LIN {X 0,Y 374.038,Z 429.773,A -85,B 0,C 180,E1 -12878.338,E2 -12878.338} C_VEL
LIN {X 0,Y 374.558,Z 418.473,A -85,B 0,C 180,E1 -12878.666,E2 -12878.666} C_VEL
LIN {X 0,Y 375.248,Z 375.181,A -85,B 0,C 180,E1 -12879.496,E2 -12879.496} C_VEL
LIN {X 0,Y 374.687,Z 369.374,A -85,B 0,C 180,E1 -12879.636,E2 -12879.636} C_VEL
LIN {X 0,Y 369.567,Z 350.642,A -85,B 0,C 180,E1 -12880.251,E2 -12880.251} C_VEL
LIN {X 0,Y 368.943,Z 344.836,A -85,B 0,C 180,E1 -12880.398,E2 -12880.398} C_VEL
LIN {X 0,Y 368.816,Z 338.494,A -85,B 0,C 180,E1 -12880.532,E2 -12880.532} C_VEL
LIN {X 0,Y 365.256,Z 319.525,A -85,B 0,C 180,E1 -12881.096,E2 -12881.096} C_VEL
LIN {X 0,Y 363.7,Z 314.51,A -85,B 0,C 180,E1 -12881.284,E2 -12881.284} C_VEL
LIN {X 0,Y 361.999,Z 305.393,A -85,B 0,C 180,E1 -12883.707,E2 -12883.707} C_VEL
LIN {X 0,Y 361.926,Z 305.399,A -85,B 0,C 180,E1 -12886.933,E2 -12886.933} C_VEL
LIN {X 0,Y 361.885,Z 305.41,A -85,B 0,C 180,E1 -12890.46,E2 -12890.46} C_VEL
LIN {X 0,Y 361.875,Z 305.406,A -85,B 0,C 180,E1 -12894.106,E2 -12894.106} C_VEL
LIN {X 0,Y 361.832,Z 305.41,A -85,B 0,C 180,E1 -12897.784,E2 -12897.784} C_VEL
LIN {X 0,Y 361.843,Z 305.41,A -85,B 0,C 180,E1 -12901.284,E2 -12901.284} C_VEL
LIN {X 0,Y 361.85,Z 305.409,A -85,B 0,C 180,E1 -12904.28,E2 -12904.28} C_VEL
LIN {X 0,Y 361.856,Z 305.41,A -85,B 0,C 180,E1 -12907.221,E2 -12907.221} C_VEL
LIN {X 0,Y 361.807,Z 305.417,A -85,B 0,C 180,E1 -12910.75,E2 -12910.75} C_VEL
LIN {X 0,Y 361.81,Z 305.413,A -85,B 0,C 180,E1 -12914.368,E2 -12914.368} C_VEL
LIN {X 0,Y 361.829,Z 305.413,A -85,B 0,C 180,E1 -12917.568,E2 -12917.568} C_VEL
LIN {X 0,Y 361.826,Z 305.414,A -85,B 0,C 180,E1 -12920.98,E2 -12920.98} C_VEL
LIN {X 0,Y 361.867,Z 305.406,A -85,B 0,C 180,E1 -12924.655,E2 -12924.655} C_VEL
LIN {X 0,Y 361.83,Z 305.41,A -85,B 0,C 180,E1 -12928.37,E2 -12928.37} C_VEL
LIN {X 0,Y 361.893,Z 305.403,A -85,B 0,C 180,E1 -12930.955,E2 -12930.955} C_VEL
LIN {X 0,Y 361.947,Z 305.401,A -85,B 0,C 180,E1 -12933.475,E2 -12933.475} C_VEL
LIN {X 0,Y 361.871,Z 305.406,A -85,B 0,C 180,E1 -12937.144,E2 -12937.144} C_VEL
LIN {X 0,Y 361.913,Z 305.399,A -85,B 0,C 180,E1 -12940.724,E2 -12940.724} C_VEL
LIN {X 0,Y 361.94,Z 305.399,A -85,B 0,C 180,E1 -12944.226,E2 -12944.226} C_VEL
LIN {X 0,Y 361.991,Z 305.391,A -85,B 0,C 180,E1 -12946.528,E2 -12946.528} C_VEL
LIN {X 0,Y 362.023,Z 305.391,A -85,B 0,C 180,E1 -12949.938,E2 -12949.938} C_VEL
LIN {X 0,Y 362.131,Z 305.372,A -85,B 0,C 180,E1 -12953.313,E2 -12953.313} C_VEL
LIN {X 0,Y 362.273,Z 305.357,A -85,B 0,C 180,E1 -12957.777,E2 -12957.777} C_VEL
LIN {X 0,Y 362.417,Z 305.34,A -85,B 0,C 180,E1 -12960,E2 -12960} C_VEL
LIN {X 0,Y 362.272,Z 305.36,A -85,B 0,C 180,E1 -12962.224,E2 -12962.224} C_VEL
LIN {X 0,Y 362.155,Z 305.374,A -85,B 0,C 180,E1 -12966.687,E2 -12966.687} C_VEL
LIN {X 0,Y 362.024,Z 305.387,A -85,B 0,C 180,E1 -12970.062,E2 -12970.062} C_VEL
LIN {X 0,Y 361.99,Z 305.39,A -85,B 0,C 180,E1 -12973.899,E2 -12973.899} C_VEL
LIN {X 0,Y 361.96,Z 305.394,A -85,B 0,C 180,E1 -12977.939,E2 -12977.939} C_VEL
LIN {X 0,Y 361.885,Z 305.403,A -85,B 0,C 180,E1 -12981.654,E2 -12981.654} C_VEL
LIN {X 0,Y 361.922,Z 305.402,A -85,B 0,C 180,E1 -12985.291,E2 -12985.291} C_VEL
LIN {X 0,Y 361.916,Z 305.399,A -85,B 0,C 180,E1 -12987.779,E2 -12987.779} C_VEL
LIN {X 0,Y 361.854,Z 305.409,A -85,B 0,C 180,E1 -12991.628,E2 -12991.628} C_VEL
LIN {X 0,Y 361.869,Z 305.411,A -85,B 0,C 180,E1 -12995.346,E2 -12995.346} C_VEL
LIN {X 0,Y 361.866,Z 305.408,A -85,B 0,C 180,E1 -12999.028,E2 -12999.028} C_VEL
LIN {X 0,Y 361.833,Z 305.41,A -85,B 0,C 180,E1 -13002.83,E2 -13002.83} C_VEL
LIN {X 0,Y 361.815,Z 305.414,A -85,B 0,C 180,E1 -13005.947,E2 -13005.947} C_VEL
LIN {X 0,Y 361.832,Z 305.412,A -85,B 0,C 180,E1 -13009.246,E2 -13009.246} C_VEL
LIN {X 0,Y 361.86,Z 305.406,A -85,B 0,C 180,E1 -13012.778,E2 -13012.778} C_VEL
LIN {X 0,Y 361.852,Z 305.413,A -85,B 0,C 180,E1 -13015.721,E2 -13015.721} C_VEL
LIN {X 0,Y 361.879,Z 305.408,A -85,B 0,C 180,E1 -13019.674,E2 -13019.674} C_VEL
LIN {X 0,Y 361.958,Z 305.54,A -85,B 0,C 180,E1 -13020.857,E2 -13020.857} C_VEL
LIN {X 0,Y 364.226,Z 316.996,A -85,B 0,C 180,E1 -13023.654,E2 -13023.654} C_VEL
LIN {X 0,Y 365.221,Z 322.463,A -85,B 0,C 180,E1 -13024.955,E2 -13024.955} C_VEL
LIN {X 0,Y 363.924,Z 338.418,A -85,B 0,C 180,E1 -13028.475,E2 -13028.475} C_VEL
LIN {X 0,Y 363.833,Z 339.649,A -85,B 0,C 180,E1 -13028.745,E2 -13028.745} C_VEL
LIN {X 0,Y 368.566,Z 373.996,A -85,B 0,C 180,E1 -13029.672,E2 -13029.672} C_VEL
LIN {X 0,Y 367.471,Z 448.258,A -85,B 0,C 180,E1 -13031.136,E2 -13031.136} C_VEL
LIN {X 0,Y 366.835,Z 461.529,A -85,B 0,C 180,E1 -13031.609,E2 -13031.609} C_VEL
LIN {X 0,Y 366.107,Z 473.727,A -85,B 0,C 180,E1 -13032.258,E2 -13032.258} C_VEL
LIN {X 0,Y 365.225,Z 485.208,A -85,B 0,C 180,E1 -13033.08,E2 -13033.08} C_VEL
LIN {X 0,Y 364.253,Z 497.008,A -85,B 0,C 180,E1 -13034.186,E2 -13034.186} C_VEL
LIN {X 0,Y 363.386,Z 507.607,A -85,B 0,C 180,E1 -13035.439,E2 -13035.439} C_VEL
LIN {X 0,Y 362.499,Z 517.133,A -85,B 0,C 180,E1 -13036.833,E2 -13036.833} C_VEL
LIN {X 0,Y 361.639,Z 526.297,A -85,B 0,C 180,E1 -13038.511,E2 -13038.511} C_VEL
LIN {X 0,Y 361.057,Z 533.678,A -85,B 0,C 180,E1 -13040.194,E2 -13040.194} C_VEL
LIN {X 0,Y 360.74,Z 538.672,A -85,B 0,C 180,E1 -13041.599,E2 -13041.599} C_VEL
LIN {X 0,Y 360.485,Z 543.511,A -85,B 0,C 180,E1 -13043.283,E2 -13043.283} C_VEL
LIN {X 0,Y 360.372,Z 547.214,A -85,B 0,C 180,E1 -13044.966,E2 -13044.966} C_VEL
LIN {X 0,Y 360.321,Z 549.885,A -85,B 0,C 180,E1 -13046.646,E2 -13046.646} C_VEL
LIN {X 0,Y 360.326,Z 551.141,A -85,B 0,C 180,E1 -13047.765,E2 -13047.765} C_VEL
LIN {X 0,Y 360.389,Z 551.991,A -85,B 0,C 180,E1 -13048.883,E2 -13048.883} C_VEL
LIN {X 0,Y 360.423,Z 552.4,A -85,B 0,C 180,E1 -13050.001,E2 -13050.001} C_VEL
LIN {X 0,Y 360.358,Z 552.415,A -85,B 0,C 180,E1 -13051.118,E2 -13051.118} C_VEL
LIN {X 0,Y 360.301,Z 551.289,A -85,B 0,C 180,E1 -13053.355,E2 -13053.355} C_VEL
LIN {X 0,Y 360.366,Z 550.094,A -85,B 0,C 180,E1 -13054.475,E2 -13054.475} C_VEL
LIN {X 0,Y 360.499,Z 546.471,A -85,B 0,C 180,E1 -13056.718,E2 -13056.718} C_VEL
LIN {X 0,Y 360.801,Z 542.572,A -85,B 0,C 180,E1 -13058.401,E2 -13058.401} C_VEL
LIN {X 0,Y 361.287,Z 537.56,A -85,B 0,C 180,E1 -13060.083,E2 -13060.083} C_VEL
LIN {X 0,Y 362.03,Z 531.286,A -85,B 0,C 180,E1 -13061.762,E2 -13061.762} C_VEL
LIN {X 0,Y 363.145,Z 523.46,A -85,B 0,C 180,E1 -13063.429,E2 -13063.429} C_VEL
LIN {X 0,Y 364.147,Z 515.494,A -85,B 0,C 180,E1 -13064.818,E2 -13064.818} C_VEL
LIN {X 0,Y 365.252,Z 505.819,A -85,B 0,C 180,E1 -13066.201,E2 -13066.201} C_VEL
LIN {X 0,Y 366.595,Z 495.078,A -85,B 0,C 180,E1 -13067.431,E2 -13067.431} C_VEL
LIN {X 0,Y 367.81,Z 484.646,A -85,B 0,C 180,E1 -13068.378,E2 -13068.378} C_VEL
LIN {X 0,Y 368.987,Z 472.123,A -85,B 0,C 180,E1 -13069.254,E2 -13069.254} C_VEL
LIN {X 0,Y 369.998,Z 458.92,A -85,B 0,C 180,E1 -13069.921,E2 -13069.921} C_VEL
LIN {X 0,Y 370.628,Z 446.91,A -85,B 0,C 180,E1 -13070.319,E2 -13070.319} C_VEL
LIN {X 0,Y 372.066,Z 375.094,A -85,B 0,C 180,E1 -13071.737,E2 -13071.737} C_VEL
LIN {X 0,Y 368.383,Z 353.004,A -85,B 0,C 180,E1 -13072.469,E2 -13072.469} C_VEL
LIN {X 0,Y 365.523,Z 339.056,A -85,B 0,C 180,E1 -13073.001,E2 -13073.001} C_VEL
LIN {X 0,Y 366.663,Z 327.943,A -85,B 0,C 180,E1 -13075.517,E2 -13075.517} C_VEL
LIN {X 0,Y 365.153,Z 319.279,A -85,B 0,C 180,E1 -13077.705,E2 -13077.705} C_VEL
LIN {X 0,Y 362.633,Z 308.581,A -85,B 0,C 180,E1 -13080.562,E2 -13080.562} C_VEL
LIN {X 0,Y 361.855,Z 305.416,A -85,B 0,C 180,E1 -13081.462,E2 -13081.462} C_VEL
LIN {X 0,Y 361.856,Z 305.415,A -85,B 0,C 180,E1 -13084.28,E2 -13084.28} C_VEL
LIN {X 0,Y 361.865,Z 305.41,A -85,B 0,C 180,E1 -13087.223,E2 -13087.223} C_VEL
LIN {X 0,Y 361.837,Z 305.414,A -85,B 0,C 180,E1 -13090.755,E2 -13090.755} C_VEL
LIN {X 0,Y 361.818,Z 305.415,A -85,B 0,C 180,E1 -13094.368,E2 -13094.368} C_VEL
LIN {X 0,Y 361.837,Z 305.41,A -85,B 0,C 180,E1 -13097.568,E2 -13097.568} C_VEL
LIN {X 0,Y 361.87,Z 305.411,A -85,B 0,C 180,E1 -13100.973,E2 -13100.973} C_VEL
LIN {X 0,Y 361.875,Z 305.409,A -85,B 0,C 180,E1 -13104.655,E2 -13104.655} C_VEL
LIN {X 0,Y 361.838,Z 305.411,A -85,B 0,C 180,E1 -13108.37,E2 -13108.37} C_VEL
LIN {X 0,Y 361.901,Z 305.404,A -85,B 0,C 180,E1 -13110.955,E2 -13110.955} C_VEL
LIN {X 0,Y 361.954,Z 305.395,A -85,B 0,C 180,E1 -13113.475,E2 -13113.475} C_VEL
LIN {X 0,Y 361.89,Z 305.402,A -85,B 0,C 180,E1 -13117.144,E2 -13117.144} C_VEL
LIN {X 0,Y 361.92,Z 305.398,A -85,B 0,C 180,E1 -13120.724,E2 -13120.724} C_VEL
LIN {X 0,Y 361.946,Z 305.394,A -85,B 0,C 180,E1 -13124.226,E2 -13124.226} C_VEL
LIN {X 0,Y 361.998,Z 305.385,A -85,B 0,C 180,E1 -13126.528,E2 -13126.528} C_VEL
LIN {X 0,Y 362.03,Z 305.38,A -85,B 0,C 180,E1 -13129.938,E2 -13129.938} C_VEL
LIN {X 0,Y 362.162,Z 305.368,A -85,B 0,C 180,E1 -13133.313,E2 -13133.313} C_VEL
LIN {X 0,Y 362.28,Z 305.353,A -85,B 0,C 180,E1 -13137.776,E2 -13137.776} C_VEL
LIN {X 0,Y 362.425,Z 305.332,A -85,B 0,C 180,E1 -13140,E2 -13140} C_VEL
LIN {X 0,Y 362.279,Z 305.351,A -85,B 0,C 180,E1 -13142.223,E2 -13142.223} C_VEL
LIN {X 0,Y 362.169,Z 305.364,A -85,B 0,C 180,E1 -13146.686,E2 -13146.686} C_VEL
LIN {X 0,Y 362.073,Z 305.379,A -85,B 0,C 180,E1 -13148.933,E2 -13148.933} C_VEL
LIN {X 0,Y 361.959,Z 305.392,A -85,B 0,C 180,E1 -13152.332,E2 -13152.332} C_VEL
LIN {X 0,Y 361.961,Z 305.398,A -85,B 0,C 180,E1 -13154.62,E2 -13154.62} C_VEL
LIN {X 0,Y 361.959,Z 305.395,A -85,B 0,C 180,E1 -13158.099,E2 -13158.099} C_VEL
LIN {X 0,Y 361.861,Z 305.405,A -85,B 0,C 180,E1 -13161.655,E2 -13161.655} C_VEL
LIN {X 0,Y 361.926,Z 305.399,A -85,B 0,C 180,E1 -13165.29,E2 -13165.29} C_VEL
LIN {X 0,Y 361.907,Z 305.396,A -85,B 0,C 180,E1 -13167.779,E2 -13167.779} C_VEL
LIN {X 0,Y 361.837,Z 305.406,A -85,B 0,C 180,E1 -13171.629,E2 -13171.629} C_VEL
LIN {X 0,Y 361.874,Z 305.406,A -85,B 0,C 180,E1 -13175.345,E2 -13175.345} C_VEL
LIN {X 0,Y 361.869,Z 305.41,A -85,B 0,C 180,E1 -13179.026,E2 -13179.026} C_VEL
LIN {X 0,Y 361.836,Z 305.411,A -85,B 0,C 180,E1 -13182.829,E2 -13182.829} C_VEL
LIN {X 0,Y 361.818,Z 305.415,A -85,B 0,C 180,E1 -13185.947,E2 -13185.947} C_VEL
LIN {X 0,Y 361.835,Z 305.414,A -85,B 0,C 180,E1 -13189.245,E2 -13189.245} C_VEL
LIN {X 0,Y 361.863,Z 305.406,A -85,B 0,C 180,E1 -13192.777,E2 -13192.777} C_VEL
LIN {X 0,Y 361.901,Z 305.436,A -85,B 0,C 180,E1 -13194.281,E2 -13194.281} C_VEL
LIN {X 0,Y 364.025,Z 314.87,A -85,B 0,C 180,E1 -13196.936,E2 -13196.936} C_VEL
LIN {X 0,Y 370.044,Z 329.595,A -85,B 0,C 180,E1 -13197.715,E2 -13197.715} C_VEL
LIN {X 0,Y 372.631,Z 341.079,A -85,B 0,C 180,E1 -13198.148,E2 -13198.148} C_VEL
LIN {X 0,Y 370.875,Z 421.936,A -85,B 0,C 180,E1 -13199.738,E2 -13199.738} C_VEL
LIN {X 0,Y 370.259,Z 434.827,A -85,B 0,C 180,E1 -13200.193,E2 -13200.193} C_VEL
LIN {X 0,Y 369.6,Z 447.003,A -85,B 0,C 180,E1 -13200.844,E2 -13200.844} C_VEL
LIN {X 0,Y 368.665,Z 458.851,A -85,B 0,C 180,E1 -13201.692,E2 -13201.692} C_VEL
LIN {X 0,Y 367.424,Z 470.91,A -85,B 0,C 180,E1 -13202.827,E2 -13202.827} C_VEL
LIN {X 0,Y 366.259,Z 481.223,A -85,B 0,C 180,E1 -13204.056,E2 -13204.056} C_VEL
LIN {X 0,Y 364.956,Z 491.237,A -85,B 0,C 180,E1 -13205.542,E2 -13205.542} C_VEL
LIN {X 0,Y 363.653,Z 500.421,A -85,B 0,C 180,E1 -13207.261,E2 -13207.261} C_VEL
LIN {X 0,Y 362.695,Z 507.766,A -85,B 0,C 180,E1 -13208.993,E2 -13208.993} C_VEL
LIN {X 0,Y 361.869,Z 513.554,A -85,B 0,C 180,E1 -13210.721,E2 -13210.721} C_VEL
LIN {X 0,Y 361.311,Z 517.926,A -85,B 0,C 180,E1 -13212.386,E2 -13212.386} C_VEL
LIN {X 0,Y 360.829,Z 521.454,A -85,B 0,C 180,E1 -13214.176,E2 -13214.176} C_VEL
LIN {X 0,Y 360.606,Z 523.12,A -85,B 0,C 180,E1 -13215.323,E2 -13215.323} C_VEL
LIN {X 0,Y 360.45,Z 524.885,A -85,B 0,C 180,E1 -13217.133,E2 -13217.133} C_VEL
LIN {X 0,Y 360.317,Z 525.591,A -85,B 0,C 180,E1 -13218.752,E2 -13218.752} C_VEL
LIN {X 0,Y 360.256,Z 525.204,A -85,B 0,C 180,E1 -13221.021,E2 -13221.021} C_VEL
LIN {X 0,Y 360.357,Z 524.401,A -85,B 0,C 180,E1 -13222.153,E2 -13222.153} C_VEL
LIN {X 0,Y 360.524,Z 522.465,A -85,B 0,C 180,E1 -13223.818,E2 -13223.818} C_VEL
LIN {X 0,Y 360.615,Z 519.498,A -85,B 0,C 180,E1 -13225.528,E2 -13225.528} C_VEL
LIN {X 0,Y 360.906,Z 515.533,A -85,B 0,C 180,E1 -13227.209,E2 -13227.209} C_VEL
LIN {X 0,Y 361.298,Z 509.444,A -85,B 0,C 180,E1 -13229.163,E2 -13229.163} C_VEL
LIN {X 0,Y 361.993,Z 502.786,A -85,B 0,C 180,E1 -13230.834,E2 -13230.834} C_VEL
LIN {X 0,Y 362.741,Z 494.551,A -85,B 0,C 180,E1 -13232.498,E2 -13232.498} C_VEL
LIN {X 0,Y 363.466,Z 486.104,A -85,B 0,C 180,E1 -13233.88,E2 -13233.88} C_VEL
LIN {X 0,Y 364.378,Z 475.674,A -85,B 0,C 180,E1 -13235.256,E2 -13235.256} C_VEL
LIN {X 0,Y 365.275,Z 466.727,A -85,B 0,C 180,E1 -13236.212,E2 -13236.212} C_VEL
LIN {X 0,Y 366.158,Z 455.721,A -85,B 0,C 180,E1 -13237.166,E2 -13237.166} C_VEL
LIN {X 0,Y 366.796,Z 443.576,A -85,B 0,C 180,E1 -13237.984,E2 -13237.984} C_VEL
LIN {X 0,Y 367.157,Z 430.842,A -85,B 0,C 180,E1 -13238.6,E2 -13238.6} C_VEL
LIN {X 0,Y 367.748,Z 418.549,A -85,B 0,C 180,E1 -13238.967,E2 -13238.967} C_VEL
LIN {X 0,Y 368.943,Z 344.836,A -85,B 0,C 180,E1 -13240.398,E2 -13240.398} C_VEL
LIN {X 0,Y 368.515,Z 340.992,A -85,B 0,C 180,E1 -13240.497,E2 -13240.497} C_VEL
LIN {X 0,Y 366.731,Z 335.502,A -85,B 0,C 180,E1 -13240.697,E2 -13240.697} C_VEL
LIN {X 0,Y 358.451,Z 320.029,A -85,B 0,C 180,E1 -13241.442,E2 -13241.442} C_VEL
LIN {X 0,Y 357.016,Z 316.361,A -85,B 0,C 180,E1 -13241.596,E2 -13241.596} C_VEL
LIN {X 0,Y 356.552,Z 314.673,A -85,B 0,C 180,E1 -13241.684,E2 -13241.684} C_VEL
LIN {X 0,Y 354.937,Z 306.273,A -85,B 0,C 180,E1 -13243.949,E2 -13243.949} C_VEL
LIN {X 0,Y 354.878,Z 306.276,A -85,B 0,C 180,E1 -13247.28,E2 -13247.28} C_VEL
LIN {X 0,Y 354.825,Z 306.285,A -85,B 0,C 180,E1 -13250.886,E2 -13250.886} C_VEL
LIN {X 0,Y 354.838,Z 306.288,A -85,B 0,C 180,E1 -13254.577,E2 -13254.577} C_VEL
LIN {X 0,Y 354.793,Z 306.29,A -85,B 0,C 180,E1 -13258.385,E2 -13258.385} C_VEL
LIN {X 0,Y 354.783,Z 306.29,A -85,B 0,C 180,E1 -13262.333,E2 -13262.333} C_VEL
LIN {X 0,Y 354.818,Z 306.283,A -85,B 0,C 180,E1 -13265.698,E2 -13265.698} C_VEL
LIN {X 0,Y 354.763,Z 306.292,A -85,B 0,C 180,E1 -13269.412,E2 -13269.412} C_VEL
LIN {X 0,Y 354.78,Z 306.293,A -85,B 0,C 180,E1 -13272.866,E2 -13272.866} C_VEL
LIN {X 0,Y 354.76,Z 306.29,A -85,B 0,C 180,E1 -13276.103,E2 -13276.103} C_VEL
LIN {X 0,Y 354.78,Z 306.294,A -85,B 0,C 180,E1 -13279.178,E2 -13279.178} C_VEL
LIN {X 0,Y 354.795,Z 306.286,A -85,B 0,C 180,E1 -13282.403,E2 -13282.403} C_VEL
LIN {X 0,Y 354.805,Z 306.287,A -85,B 0,C 180,E1 -13284.94,E2 -13284.94} C_VEL
LIN {X 0,Y 354.786,Z 306.287,A -85,B 0,C 180,E1 -13288.405,E2 -13288.405} C_VEL
LIN {X 0,Y 354.844,Z 306.286,A -85,B 0,C 180,E1 -13291.619,E2 -13291.619} C_VEL
LIN {X 0,Y 354.89,Z 306.276,A -85,B 0,C 180,E1 -13294.172,E2 -13294.172} C_VEL
LIN {X 0,Y 354.808,Z 306.289,A -85,B 0,C 180,E1 -13297.892,E2 -13297.892} C_VEL
LIN {X 0,Y 354.915,Z 306.277,A -85,B 0,C 180,E1 -13301.891,E2 -13301.891} C_VEL
LIN {X 0,Y 354.935,Z 306.275,A -85,B 0,C 180,E1 -13305.981,E2 -13305.981} C_VEL
LIN {X 0,Y 354.969,Z 306.268,A -85,B 0,C 180,E1 -13309.736,E2 -13309.736} C_VEL
LIN {X 0,Y 355.094,Z 306.249,A -85,B 0,C 180,E1 -13313.18,E2 -13313.18} C_VEL
LIN {X 0,Y 355.236,Z 306.233,A -85,B 0,C 180,E1 -13317.732,E2 -13317.732} C_VEL
LIN {X 0,Y 355.366,Z 306.218,A -85,B 0,C 180,E1 -13320,E2 -13320} C_VEL
LIN {X 0,Y 355.235,Z 306.237,A -85,B 0,C 180,E1 -13322.268,E2 -13322.268} C_VEL
LIN {X 0,Y 355.119,Z 306.249,A -85,B 0,C 180,E1 -13326.82,E2 -13326.82} C_VEL
LIN {X 0,Y 354.97,Z 306.267,A -85,B 0,C 180,E1 -13330.264,E2 -13330.264} C_VEL
LIN {X 0,Y 354.935,Z 306.269,A -85,B 0,C 180,E1 -13334.019,E2 -13334.019} C_VEL
LIN {X 0,Y 354.915,Z 306.272,A -85,B 0,C 180,E1 -13338.109,E2 -13338.109} C_VEL
LIN {X 0,Y 354.828,Z 306.282,A -85,B 0,C 180,E1 -13342.107,E2 -13342.107} C_VEL
LIN {X 0,Y 354.893,Z 306.274,A -85,B 0,C 180,E1 -13345.828,E2 -13345.828} C_VEL
LIN {X 0,Y 354.849,Z 306.281,A -85,B 0,C 180,E1 -13349.679,E2 -13349.679} C_VEL
LIN {X 0,Y 354.825,Z 306.284,A -85,B 0,C 180,E1 -13353.683,E2 -13353.683} C_VEL
LIN {X 0,Y 354.796,Z 306.286,A -85,B 0,C 180,E1 -13356.46,E2 -13356.46} C_VEL
LIN {X 0,Y 354.819,Z 306.289,A -85,B 0,C 180,E1 -13359.425,E2 -13359.425} C_VEL
LIN {X 0,Y 354.785,Z 306.289,A -85,B 0,C 180,E1 -13362.868,E2 -13362.868} C_VEL
LIN {X 0,Y 354.764,Z 306.291,A -85,B 0,C 180,E1 -13366.105,E2 -13366.105} C_VEL
LIN {X 0,Y 354.784,Z 306.29,A -85,B 0,C 180,E1 -13369.18,E2 -13369.18} C_VEL
LIN {X 0,Y 354.804,Z 306.286,A -85,B 0,C 180,E1 -13372.404,E2 -13372.404} C_VEL
LIN {X 0,Y 354.809,Z 306.285,A -85,B 0,C 180,E1 -13374.942,E2 -13374.942} C_VEL
LIN {X 0,Y 354.792,Z 306.288,A -85,B 0,C 180,E1 -13378.406,E2 -13378.406} C_VEL
LIN {X 0,Y 354.867,Z 306.307,A -85,B 0,C 180,E1 -13380.554,E2 -13380.554} C_VEL
LIN {X 0,Y 357.173,Z 317.74,A -85,B 0,C 180,E1 -13383.408,E2 -13383.408} C_VEL
LIN {X 0,Y 358.182,Z 323.116,A -85,B 0,C 180,E1 -13384.717,E2 -13384.717} C_VEL
LIN {X 0,Y 357.511,Z 332.543,A -85,B 0,C 180,E1 -13386.85,E2 -13386.85} C_VEL
LIN {X 0,Y 356.906,Z 339.368,A -85,B 0,C 180,E1 -13388.378,E2 -13388.378} C_VEL
LIN {X 0,Y 361.785,Z 374.313,A -85,B 0,C 180,E1 -13389.351,E2 -13389.351} C_VEL
LIN {X 0,Y 360.643,Z 448.305,A -85,B 0,C 180,E1 -13390.839,E2 -13390.839} C_VEL
LIN {X 0,Y 359.949,Z 462.24,A -85,B 0,C 180,E1 -13391.355,E2 -13391.355} C_VEL
LIN {X 0,Y 359.169,Z 474.728,A -85,B 0,C 180,E1 -13392.051,E2 -13392.051} C_VEL
LIN {X 0,Y 358.14,Z 487.459,A -85,B 0,C 180,E1 -13393.029,E2 -13393.029} C_VEL
LIN {X 0,Y 357.162,Z 498.792,A -85,B 0,C 180,E1 -13394.157,E2 -13394.157} C_VEL
LIN {X 0,Y 356.282,Z 508.981,A -85,B 0,C 180,E1 -13395.434,E2 -13395.434} C_VEL
LIN {X 0,Y 355.399,Z 518.164,A -85,B 0,C 180,E1 -13396.856,E2 -13396.856} C_VEL
LIN {X 0,Y 354.499,Z 527.105,A -85,B 0,C 180,E1 -13398.566,E2 -13398.566} C_VEL
LIN {X 0,Y 353.948,Z 534.277,A -85,B 0,C 180,E1 -13400.284,E2 -13400.284} C_VEL
LIN {X 0,Y 353.55,Z 539.983,A -85,B 0,C 180,E1 -13402.002,E2 -13402.002} C_VEL
LIN {X 0,Y 353.322,Z 545.136,A -85,B 0,C 180,E1 -13404.024,E2 -13404.024} C_VEL
LIN {X 0,Y 353.29,Z 547.863,A -85,B 0,C 180,E1 -13405.437,E2 -13405.437} C_VEL
LIN {X 0,Y 353.241,Z 549.542,A -85,B 0,C 180,E1 -13406.579,E2 -13406.579} C_VEL
LIN {X 0,Y 353.291,Z 551.691,A -85,B 0,C 180,E1 -13408.861,E2 -13408.861} C_VEL
LIN {X 0,Y 353.328,Z 552.126,A -85,B 0,C 180,E1 -13410.001,E2 -13410.001} C_VEL
LIN {X 0,Y 353.26,Z 552.159,A -85,B 0,C 180,E1 -13411.141,E2 -13411.141} C_VEL
LIN {X 0,Y 353.223,Z 551.071,A -85,B 0,C 180,E1 -13413.423,E2 -13413.423} C_VEL
LIN {X 0,Y 353.279,Z 549.906,A -85,B 0,C 180,E1 -13414.565,E2 -13414.565} C_VEL
LIN {X 0,Y 353.317,Z 547.907,A -85,B 0,C 180,E1 -13415.968,E2 -13415.968} C_VEL
LIN {X 0,Y 353.617,Z 543.886,A -85,B 0,C 180,E1 -13417.998,E2 -13417.998} C_VEL
LIN {X 0,Y 354.062,Z 539.299,A -85,B 0,C 180,E1 -13419.714,E2 -13419.714} C_VEL
LIN {X 0,Y 354.908,Z 532.378,A -85,B 0,C 180,E1 -13421.711,E2 -13421.711} C_VEL
LIN {X 0,Y 356.015,Z 524.91,A -85,B 0,C 180,E1 -13423.413,E2 -13423.413} C_VEL
LIN {X 0,Y 357.226,Z 515.93,A -85,B 0,C 180,E1 -13425.06,E2 -13425.06} C_VEL
LIN {X 0,Y 358.43,Z 506.023,A -85,B 0,C 180,E1 -13426.518,E2 -13426.518} C_VEL
LIN {X 0,Y 359.856,Z 495.385,A -85,B 0,C 180,E1 -13427.768,E2 -13427.768} C_VEL
LIN {X 0,Y 361.101,Z 485.113,A -85,B 0,C 180,E1 -13428.732,E2 -13428.732} C_VEL
LIN {X 0,Y 362.326,Z 472.876,A -85,B 0,C 180,E1 -13429.622,E2 -13429.622} C_VEL
LIN {X 0,Y 363.391,Z 460.031,A -85,B 0,C 180,E1 -13430.299,E2 -13430.299} C_VEL
LIN {X 0,Y 364.071,Z 447.666,A -85,B 0,C 180,E1 -13430.739,E2 -13430.739} C_VEL
LIN {X 0,Y 365.542,Z 375.302,A -85,B 0,C 180,E1 -13432.204,E2 -13432.204} C_VEL
LIN {X 0,Y 362.003,Z 354.385,A -85,B 0,C 180,E1 -13432.921,E2 -13432.921} C_VEL
LIN {X 0,Y 358.781,Z 338.808,A -85,B 0,C 180,E1 -13433.526,E2 -13433.526} C_VEL
LIN {X 0,Y 359.806,Z 329.05,A -85,B 0,C 180,E1 -13435.781,E2 -13435.781} C_VEL
LIN {X 0,Y 357.826,Z 318.845,A -85,B 0,C 180,E1 -13438.444,E2 -13438.444} C_VEL
LIN {X 0,Y 355.205,Z 307.939,A -85,B 0,C 180,E1 -13441.456,E2 -13441.456} C_VEL
LIN {X 0,Y 354.783,Z 306.296,A -85,B 0,C 180,E1 -13441.967,E2 -13441.967} C_VEL
LIN {X 0,Y 354.814,Z 306.288,A -85,B 0,C 180,E1 -13445.059,E2 -13445.059} C_VEL
LIN {X 0,Y 354.807,Z 306.291,A -85,B 0,C 180,E1 -13447.883,E2 -13447.883} C_VEL
LIN {X 0,Y 354.789,Z 306.291,A -85,B 0,C 180,E1 -13451.171,E2 -13451.171} C_VEL
LIN {X 0,Y 354.764,Z 306.293,A -85,B 0,C 180,E1 -13454.506,E2 -13454.506} C_VEL
LIN {X 0,Y 354.795,Z 306.287,A -85,B 0,C 180,E1 -13457.662,E2 -13457.662} C_VEL
LIN {X 0,Y 354.816,Z 306.285,A -85,B 0,C 180,E1 -13460.666,E2 -13460.666} C_VEL
LIN {X 0,Y 354.822,Z 306.284,A -85,B 0,C 180,E1 -13464.301,E2 -13464.301} C_VEL
LIN {X 0,Y 354.787,Z 306.289,A -85,B 0,C 180,E1 -13467.666,E2 -13467.666} C_VEL
LIN {X 0,Y 354.869,Z 306.277,A -85,B 0,C 180,E1 -13470.621,E2 -13470.621} C_VEL
LIN {X 0,Y 354.899,Z 306.273,A -85,B 0,C 180,E1 -13474.172,E2 -13474.172} C_VEL
LIN {X 0,Y 354.835,Z 306.282,A -85,B 0,C 180,E1 -13477.894,E2 -13477.894} C_VEL
LIN {X 0,Y 354.923,Z 306.27,A -85,B 0,C 180,E1 -13481.891,E2 -13481.891} C_VEL
LIN {X 0,Y 354.942,Z 306.265,A -85,B 0,C 180,E1 -13485.981,E2 -13485.981} C_VEL
LIN {X 0,Y 354.977,Z 306.259,A -85,B 0,C 180,E1 -13489.736,E2 -13489.736} C_VEL
LIN {X 0,Y 355.125,Z 306.243,A -85,B 0,C 180,E1 -13493.18,E2 -13493.18} C_VEL
LIN {X 0,Y 355.243,Z 306.23,A -85,B 0,C 180,E1 -13497.732,E2 -13497.732} C_VEL
LIN {X 0,Y 355.374,Z 306.21,A -85,B 0,C 180,E1 -13500,E2 -13500} C_VEL
LIN {X 0,Y 355.242,Z 306.227,A -85,B 0,C 180,E1 -13502.267,E2 -13502.267} C_VEL
LIN {X 0,Y 355.136,Z 306.239,A -85,B 0,C 180,E1 -13506.819,E2 -13506.819} C_VEL
LIN {X 0,Y 355.014,Z 306.257,A -85,B 0,C 180,E1 -13509.112,E2 -13509.112} C_VEL
LIN {X 0,Y 354.92,Z 306.269,A -85,B 0,C 180,E1 -13512.581,E2 -13512.581} C_VEL
LIN {X 0,Y 354.889,Z 306.275,A -85,B 0,C 180,E1 -13516.096,E2 -13516.096} C_VEL
LIN {X 0,Y 354.906,Z 306.277,A -85,B 0,C 180,E1 -13518.472,E2 -13518.472} C_VEL
LIN {X 0,Y 354.816,Z 306.284,A -85,B 0,C 180,E1 -13522.107,E2 -13522.107} C_VEL
LIN {X 0,Y 354.898,Z 306.273,A -85,B 0,C 180,E1 -13525.827,E2 -13525.827} C_VEL
LIN {X 0,Y 354.817,Z 306.283,A -85,B 0,C 180,E1 -13529.682,E2 -13529.682} C_VEL
LIN {X 0,Y 354.806,Z 306.284,A -85,B 0,C 180,E1 -13533.702,E2 -13533.702} C_VEL
LIN {X 0,Y 354.797,Z 306.288,A -85,B 0,C 180,E1 -13536.459,E2 -13536.459} C_VEL
LIN {X 0,Y 354.824,Z 306.285,A -85,B 0,C 180,E1 -13539.424,E2 -13539.424} C_VEL
LIN {X 0,Y 354.788,Z 306.289,A -85,B 0,C 180,E1 -13542.867,E2 -13542.867} C_VEL
LIN {X 0,Y 354.767,Z 306.293,A -85,B 0,C 180,E1 -13546.104,E2 -13546.104} C_VEL
LIN {X 0,Y 354.788,Z 306.292,A -85,B 0,C 180,E1 -13549.179,E2 -13549.179} C_VEL
LIN {X 0,Y 354.807,Z 306.283,A -85,B 0,C 180,E1 -13552.403,E2 -13552.403} C_VEL
LIN {X 0,Y 354.852,Z 306.332,A -85,B 0,C 180,E1 -13553.81,E2 -13553.81} C_VEL
LIN {X 0,Y 356.907,Z 315.288,A -85,B 0,C 180,E1 -13556.369,E2 -13556.369} C_VEL
LIN {X 0,Y 363.679,Z 331.28,A -85,B 0,C 180,E1 -13557.265,E2 -13557.265} C_VEL
LIN {X 0,Y 366.185,Z 342.113,A -85,B 0,C 180,E1 -13557.69,E2 -13557.69} C_VEL
LIN {X 0,Y 364.392,Z 422.475,A -85,B 0,C 180,E1 -13559.303,E2 -13559.303} C_VEL
LIN {X 0,Y 363.679,Z 436.04,A -85,B 0,C 180,E1 -13559.798,E2 -13559.798} C_VEL
LIN {X 0,Y 362.969,Z 448.613,A -85,B 0,C 180,E1 -13560.501,E2 -13560.501} C_VEL
LIN {X 0,Y 361.896,Z 460.862,A -85,B 0,C 180,E1 -13561.431,E2 -13561.431} C_VEL
LIN {X 0,Y 360.638,Z 472.576,A -85,B 0,C 180,E1 -13562.587,E2 -13562.587} C_VEL
LIN {X 0,Y 359.373,Z 482.784,A -85,B 0,C 180,E1 -13563.856,E2 -13563.856} C_VEL
LIN {X 0,Y 358.043,Z 492.37,A -85,B 0,C 180,E1 -13565.347,E2 -13565.347} C_VEL
LIN {X 0,Y 356.698,Z 501.403,A -85,B 0,C 180,E1 -13567.099,E2 -13567.099} C_VEL
LIN {X 0,Y 355.697,Z 508.603,A -85,B 0,C 180,E1 -13568.873,E2 -13568.873} C_VEL
LIN {X 0,Y 354.718,Z 515.061,A -85,B 0,C 180,E1 -13570.918,E2 -13570.918} C_VEL
LIN {X 0,Y 354.136,Z 519.287,A -85,B 0,C 180,E1 -13572.681,E2 -13572.681} C_VEL
LIN {X 0,Y 353.834,Z 521.5,A -85,B 0,C 180,E1 -13573.854,E2 -13573.854} C_VEL
LIN {X 0,Y 353.564,Z 523.209,A -85,B 0,C 180,E1 -13575.024,E2 -13575.024} C_VEL
LIN {X 0,Y 353.389,Z 525.161,A -85,B 0,C 180,E1 -13577.029,E2 -13577.029} C_VEL
LIN {X 0,Y 353.232,Z 525.839,A -85,B 0,C 180,E1 -13578.523,E2 -13578.523} C_VEL
LIN {X 0,Y 353.153,Z 525.529,A -85,B 0,C 180,E1 -13580.839,E2 -13580.839} C_VEL
LIN {X 0,Y 353.257,Z 524.789,A -85,B 0,C 180,E1 -13581.994,E2 -13581.994} C_VEL
LIN {X 0,Y 353.43,Z 522.697,A -85,B 0,C 180,E1 -13583.856,E2 -13583.856} C_VEL
LIN {X 0,Y 353.553,Z 518.84,A -85,B 0,C 180,E1 -13586.01,E2 -13586.01} C_VEL
LIN {X 0,Y 353.925,Z 514.595,A -85,B 0,C 180,E1 -13587.723,E2 -13587.723} C_VEL
LIN {X 0,Y 354.45,Z 508.18,A -85,B 0,C 180,E1 -13589.715,E2 -13589.715} C_VEL
LIN {X 0,Y 355.153,Z 501.148,A -85,B 0,C 180,E1 -13591.417,E2 -13591.417} C_VEL
LIN {X 0,Y 355.979,Z 492.39,A -85,B 0,C 180,E1 -13593.112,E2 -13593.112} C_VEL
LIN {X 0,Y 356.854,Z 482.456,A -85,B 0,C 180,E1 -13594.659,E2 -13594.659} C_VEL
LIN {X 0,Y 357.79,Z 472.286,A -85,B 0,C 180,E1 -13595.918,E2 -13595.918} C_VEL
LIN {X 0,Y 358.854,Z 462.522,A -85,B 0,C 180,E1 -13596.889,E2 -13596.889} C_VEL
LIN {X 0,Y 359.604,Z 450.278,A -85,B 0,C 180,E1 -13597.862,E2 -13597.862} C_VEL
LIN {X 0,Y 360.161,Z 438.668,A -85,B 0,C 180,E1 -13598.556,E2 -13598.556} C_VEL
LIN {X 0,Y 360.551,Z 427.29,A -85,B 0,C 180,E1 -13599.041,E2 -13599.041} C_VEL
LIN {X 0,Y 361.044,Z 413.744,A -85,B 0,C 180,E1 -13599.382,E2 -13599.382} C_VEL
LIN {X 0,Y 362.171,Z 340.065,A -85,B 0,C 180,E1 -13600.834,E2 -13600.834} C_VEL
LIN {X 0,Y 358.638,Z 321.225,A -85,B 0,C 180,E1 -13601.407,E2 -13601.407} C_VEL
LIN {X 0,Y 357.016,Z 316.361,A -85,B 0,C 180,E1 -13601.596,E2 -13601.596} C_VEL
LIN {X 0,Y 355.965,Z 314.814,A -85,B 0,C 180,E1 -13601.754,E2 -13601.754} C_VEL
LIN {X 0,Y 350.904,Z 311.687,A -85,B 0,C 180,E1 -13602.814,E2 -13602.814} C_VEL
LIN {X 0,Y 349.011,Z 309.812,A -85,B 0,C 180,E1 -13603.422,E2 -13603.422} C_VEL
LIN {X 0,Y 347.909,Z 307.271,A -85,B 0,C 180,E1 -13604.212,E2 -13604.212} C_VEL
LIN {X 0,Y 347.882,Z 307.153,A -85,B 0,C 180,E1 -13604.342,E2 -13604.342} C_VEL
LIN {X 0,Y 347.827,Z 307.159,A -85,B 0,C 180,E1 -13608.258,E2 -13608.258} C_VEL
LIN {X 0,Y 347.765,Z 307.162,A -85,B 0,C 180,E1 -13611.625,E2 -13611.625} C_VEL
LIN {X 0,Y 347.757,Z 307.164,A -85,B 0,C 180,E1 -13615.112,E2 -13615.112} C_VEL
LIN {X 0,Y 347.741,Z 307.168,A -85,B 0,C 180,E1 -13619.015,E2 -13619.015} C_VEL
LIN {X 0,Y 347.735,Z 307.166,A -85,B 0,C 180,E1 -13621.913,E2 -13621.913} C_VEL
LIN {X 0,Y 347.784,Z 307.16,A -85,B 0,C 180,E1 -13625.874,E2 -13625.874} C_VEL
LIN {X 0,Y 347.726,Z 307.172,A -85,B 0,C 180,E1 -13628.795,E2 -13628.795} C_VEL
LIN {X 0,Y 347.738,Z 307.165,A -85,B 0,C 180,E1 -13631.831,E2 -13631.831} C_VEL
LIN {X 0,Y 347.699,Z 307.176,A -85,B 0,C 180,E1 -13635.026,E2 -13635.026} C_VEL
LIN {X 0,Y 347.743,Z 307.165,A -85,B 0,C 180,E1 -13638.397,E2 -13638.397} C_VEL
LIN {X 0,Y 347.758,Z 307.163,A -85,B 0,C 180,E1 -13642.013,E2 -13642.013} C_VEL
LIN {X 0,Y 347.738,Z 307.17,A -85,B 0,C 180,E1 -13645.535,E2 -13645.535} C_VEL
LIN {X 0,Y 347.757,Z 307.168,A -85,B 0,C 180,E1 -13649.653,E2 -13649.653} C_VEL
LIN {X 0,Y 347.844,Z 307.152,A -85,B 0,C 180,E1 -13652.744,E2 -13652.744} C_VEL
LIN {X 0,Y 347.777,Z 307.162,A -85,B 0,C 180,E1 -13656.161,E2 -13656.161} C_VEL
LIN {X 0,Y 347.804,Z 307.162,A -85,B 0,C 180,E1 -13659.909,E2 -13659.909} C_VEL
LIN {X 0,Y 347.859,Z 307.152,A -85,B 0,C 180,E1 -13662.359,E2 -13662.359} C_VEL
LIN {X 0,Y 347.89,Z 307.153,A -85,B 0,C 180,E1 -13665.971,E2 -13665.971} C_VEL
LIN {X 0,Y 347.92,Z 307.144,A -85,B 0,C 180,E1 -13669.525,E2 -13669.525} C_VEL
LIN {X 0,Y 348.062,Z 307.125,A -85,B 0,C 180,E1 -13673.042,E2 -13673.042} C_VEL
LIN {X 0,Y 348.198,Z 307.109,A -85,B 0,C 180,E1 -13677.687,E2 -13677.687} C_VEL
LIN {X 0,Y 348.316,Z 307.096,A -85,B 0,C 180,E1 -13680,E2 -13680} C_VEL
LIN {X 0,Y 348.198,Z 307.114,A -85,B 0,C 180,E1 -13682.314,E2 -13682.314} C_VEL
LIN {X 0,Y 348.085,Z 307.124,A -85,B 0,C 180,E1 -13686.958,E2 -13686.958} C_VEL
LIN {X 0,Y 347.921,Z 307.148,A -85,B 0,C 180,E1 -13690.475,E2 -13690.475} C_VEL
LIN {X 0,Y 347.891,Z 307.148,A -85,B 0,C 180,E1 -13694.15,E2 -13694.15} C_VEL
LIN {X 0,Y 347.883,Z 307.149,A -85,B 0,C 180,E1 -13698.291,E2 -13698.291} C_VEL
LIN {X 0,Y 347.782,Z 307.16,A -85,B 0,C 180,E1 -13701.636,E2 -13701.636} C_VEL
LIN {X 0,Y 347.806,Z 307.162,A -85,B 0,C 180,E1 -13705.109,E2 -13705.109} C_VEL
LIN {X 0,Y 347.806,Z 307.158,A -85,B 0,C 180,E1 -13707.694,E2 -13707.694} C_VEL
LIN {X 0,Y 347.765,Z 307.162,A -85,B 0,C 180,E1 -13710.347,E2 -13710.347} C_VEL
LIN {X 0,Y 347.743,Z 307.165,A -85,B 0,C 180,E1 -13714.045,E2 -13714.045} C_VEL
LIN {X 0,Y 347.761,Z 307.169,A -85,B 0,C 180,E1 -13717.321,E2 -13717.321} C_VEL
LIN {X 0,Y 347.728,Z 307.167,A -85,B 0,C 180,E1 -13720.298,E2 -13720.298} C_VEL
LIN {X 0,Y 347.719,Z 307.174,A -85,B 0,C 180,E1 -13723.409,E2 -13723.409} C_VEL
LIN {X 0,Y 347.722,Z 307.167,A -85,B 0,C 180,E1 -13726.687,E2 -13726.687} C_VEL
LIN {X 0,Y 347.744,Z 307.166,A -85,B 0,C 180,E1 -13730.174,E2 -13730.174} C_VEL
LIN {X 0,Y 347.758,Z 307.163,A -85,B 0,C 180,E1 -13732.68,E2 -13732.68} C_VEL
LIN {X 0,Y 347.746,Z 307.169,A -85,B 0,C 180,E1 -13735.957,E2 -13735.957} C_VEL
LIN {X 0,Y 347.821,Z 307.16,A -85,B 0,C 180,E1 -13740.239,E2 -13740.239} C_VEL
LIN {X 0,Y 350.135,Z 318.466,A -85,B 0,C 180,E1 -13743.153,E2 -13743.153} C_VEL
LIN {X 0,Y 351.244,Z 324.897,A -85,B 0,C 180,E1 -13744.744,E2 -13744.744} C_VEL
LIN {X 0,Y 350.028,Z 339.056,A -85,B 0,C 180,E1 -13747.993,E2 -13747.993} C_VEL
LIN {X 0,Y 355.038,Z 375.372,A -85,B 0,C 180,E1 -13749.036,E2 -13749.036} C_VEL
LIN {X 0,Y 353.832,Z 448.266,A -85,B 0,C 180,E1 -13750.531,E2 -13750.531} C_VEL
LIN {X 0,Y 353.104,Z 462.128,A -85,B 0,C 180,E1 -13751.055,E2 -13751.055} C_VEL
LIN {X 0,Y 352.305,Z 474.572,A -85,B 0,C 180,E1 -13751.764,E2 -13751.764} C_VEL
LIN {X 0,Y 351.278,Z 486.479,A -85,B 0,C 180,E1 -13752.687,E2 -13752.687} C_VEL
LIN {X 0,Y 350.254,Z 498.077,A -85,B 0,C 180,E1 -13753.851,E2 -13753.851} C_VEL
LIN {X 0,Y 349.382,Z 507.776,A -85,B 0,C 180,E1 -13755.068,E2 -13755.068} C_VEL
LIN {X 0,Y 348.401,Z 517.538,A -85,B 0,C 180,E1 -13756.587,E2 -13756.587} C_VEL
LIN {X 0,Y 347.665,Z 525.178,A -85,B 0,C 180,E1 -13758.042,E2 -13758.042} C_VEL
LIN {X 0,Y 346.988,Z 532.662,A -85,B 0,C 180,E1 -13759.793,E2 -13759.793} C_VEL
LIN {X 0,Y 346.502,Z 539.544,A -85,B 0,C 180,E1 -13761.838,E2 -13761.838} C_VEL
LIN {X 0,Y 346.271,Z 544.197,A -85,B 0,C 180,E1 -13763.65,E2 -13763.65} C_VEL
LIN {X 0,Y 346.205,Z 547.502,A -85,B 0,C 180,E1 -13765.343,E2 -13765.343} C_VEL
LIN {X 0,Y 346.164,Z 549.2,A -85,B 0,C 180,E1 -13766.509,E2 -13766.509} C_VEL
LIN {X 0,Y 346.193,Z 551.385,A -85,B 0,C 180,E1 -13768.837,E2 -13768.837} C_VEL
LIN {X 0,Y 346.233,Z 551.853,A -85,B 0,C 180,E1 -13770.001,E2 -13770.001} C_VEL
LIN {X 0,Y 346.161,Z 551.902,A -85,B 0,C 180,E1 -13771.164,E2 -13771.164} C_VEL
LIN {X 0,Y 346.147,Z 550.849,A -85,B 0,C 180,E1 -13773.493,E2 -13773.493} C_VEL
LIN {X 0,Y 346.177,Z 549.717,A -85,B 0,C 180,E1 -13774.659,E2 -13774.659} C_VEL
LIN {X 0,Y 346.243,Z 547.944,A -85,B 0,C 180,E1 -13775.957,E2 -13775.957} C_VEL
LIN {X 0,Y 346.557,Z 543.761,A -85,B 0,C 180,E1 -13778.162,E2 -13778.162} C_VEL
LIN {X 0,Y 347.043,Z 539.218,A -85,B 0,C 180,E1 -13779.912,E2 -13779.912} C_VEL
LIN {X 0,Y 347.946,Z 532.362,A -85,B 0,C 180,E1 -13781.949,E2 -13781.949} C_VEL
LIN {X 0,Y 349.103,Z 524.951,A -85,B 0,C 180,E1 -13783.683,E2 -13783.683} C_VEL
LIN {X 0,Y 350.309,Z 516.344,A -85,B 0,C 180,E1 -13785.315,E2 -13785.315} C_VEL
LIN {X 0,Y 351.632,Z 506.243,A -85,B 0,C 180,E1 -13786.847,E2 -13786.847} C_VEL
LIN {X 0,Y 353.127,Z 495.705,A -85,B 0,C 180,E1 -13788.118,E2 -13788.118} C_VEL
LIN {X 0,Y 354.575,Z 483.956,A -85,B 0,C 180,E1 -13789.24,E2 -13789.24} C_VEL
LIN {X 0,Y 355.912,Z 471.386,A -85,B 0,C 180,E1 -13790.141,E2 -13790.141} C_VEL
LIN {X 0,Y 356.955,Z 458.875,A -85,B 0,C 180,E1 -13790.795,E2 -13790.795} C_VEL
LIN {X 0,Y 357.693,Z 445.859,A -85,B 0,C 180,E1 -13791.24,E2 -13791.24} C_VEL
LIN {X 0,Y 359.094,Z 375.72,A -85,B 0,C 180,E1 -13792.68,E2 -13792.68} C_VEL
LIN {X 0,Y 355.567,Z 355.359,A -85,B 0,C 180,E1 -13793.405,E2 -13793.405} C_VEL
LIN {X 0,Y 352.094,Z 338.431,A -85,B 0,C 180,E1 -13794.101,E2 -13794.101} C_VEL
LIN {X 0,Y 352.904,Z 330.472,A -85,B 0,C 180,E1 -13795.985,E2 -13795.985} C_VEL
LIN {X 0,Y 350.911,Z 320.185,A -85,B 0,C 180,E1 -13798.729,E2 -13798.729} C_VEL
LIN {X 0,Y 348.094,Z 308.639,A -85,B 0,C 180,E1 -13802.007,E2 -13802.007} C_VEL
LIN {X 0,Y 347.756,Z 307.166,A -85,B 0,C 180,E1 -13802.44,E2 -13802.44} C_VEL
LIN {X 0,Y 347.772,Z 307.168,A -85,B 0,C 180,E1 -13806.065,E2 -13806.065} C_VEL
LIN {X 0,Y 347.754,Z 307.168,A -85,B 0,C 180,E1 -13808.793,E2 -13808.793} C_VEL
LIN {X 0,Y 347.752,Z 307.168,A -85,B 0,C 180,E1 -13811.83,E2 -13811.83} C_VEL
LIN {X 0,Y 347.707,Z 307.173,A -85,B 0,C 180,E1 -13815.027,E2 -13815.027} C_VEL
LIN {X 0,Y 347.751,Z 307.168,A -85,B 0,C 180,E1 -13818.397,E2 -13818.397} C_VEL
LIN {X 0,Y 347.774,Z 307.162,A -85,B 0,C 180,E1 -13822.011,E2 -13822.011} C_VEL
LIN {X 0,Y 347.745,Z 307.162,A -85,B 0,C 180,E1 -13825.536,E2 -13825.536} C_VEL
LIN {X 0,Y 347.764,Z 307.16,A -85,B 0,C 180,E1 -13829.653,E2 -13829.653} C_VEL
LIN {X 0,Y 347.851,Z 307.153,A -85,B 0,C 180,E1 -13832.745,E2 -13832.745} C_VEL
LIN {X 0,Y 347.789,Z 307.159,A -85,B 0,C 180,E1 -13836.162,E2 -13836.162} C_VEL
LIN {X 0,Y 347.817,Z 307.156,A -85,B 0,C 180,E1 -13839.909,E2 -13839.909} C_VEL
LIN {X 0,Y 347.866,Z 307.148,A -85,B 0,C 180,E1 -13842.359,E2 -13842.359} C_VEL
LIN {X 0,Y 347.897,Z 307.142,A -85,B 0,C 180,E1 -13845.971,E2 -13845.971} C_VEL
LIN {X 0,Y 347.928,Z 307.138,A -85,B 0,C 180,E1 -13849.525,E2 -13849.525} C_VEL
LIN {X 0,Y 348.091,Z 307.119,A -85,B 0,C 180,E1 -13853.042,E2 -13853.042} C_VEL
LIN {X 0,Y 348.205,Z 307.106,A -85,B 0,C 180,E1 -13857.686,E2 -13857.686} C_VEL
LIN {X 0,Y 348.324,Z 307.088,A -85,B 0,C 180,E1 -13860,E2 -13860} C_VEL
LIN {X 0,Y 348.205,Z 307.103,A -85,B 0,C 180,E1 -13862.313,E2 -13862.313} C_VEL
LIN {X 0,Y 348.104,Z 307.115,A -85,B 0,C 180,E1 -13866.958,E2 -13866.958} C_VEL
LIN {X 0,Y 347.927,Z 307.144,A -85,B 0,C 180,E1 -13870.474,E2 -13870.474} C_VEL
LIN {X 0,Y 347.898,Z 307.148,A -85,B 0,C 180,E1 -13874.15,E2 -13874.15} C_VEL
LIN {X 0,Y 347.891,Z 307.149,A -85,B 0,C 180,E1 -13878.29,E2 -13878.29} C_VEL
LIN {X 0,Y 347.767,Z 307.161,A -85,B 0,C 180,E1 -13881.626,E2 -13881.626} C_VEL
LIN {X 0,Y 347.811,Z 307.156,A -85,B 0,C 180,E1 -13885.108,E2 -13885.108} C_VEL
LIN {X 0,Y 347.808,Z 307.153,A -85,B 0,C 180,E1 -13887.694,E2 -13887.694} C_VEL
LIN {X 0,Y 347.749,Z 307.165,A -85,B 0,C 180,E1 -13890.348,E2 -13890.348} C_VEL
LIN {X 0,Y 347.748,Z 307.163,A -85,B 0,C 180,E1 -13894.044,E2 -13894.044} C_VEL
LIN {X 0,Y 347.761,Z 307.163,A -85,B 0,C 180,E1 -13897.321,E2 -13897.321} C_VEL
LIN {X 0,Y 347.732,Z 307.164,A -85,B 0,C 180,E1 -13900.297,E2 -13900.297} C_VEL
LIN {X 0,Y 347.723,Z 307.172,A -85,B 0,C 180,E1 -13903.408,E2 -13903.408} C_VEL
LIN {X 0,Y 347.725,Z 307.169,A -85,B 0,C 180,E1 -13906.686,E2 -13906.686} C_VEL
LIN {X 0,Y 347.747,Z 307.168,A -85,B 0,C 180,E1 -13910.173,E2 -13910.173} C_VEL
LIN {X 0,Y 347.79,Z 307.328,A -85,B 0,C 180,E1 -13913.344,E2 -13913.344} C_VEL
LIN {X 0,Y 349.727,Z 315.435,A -85,B 0,C 180,E1 -13915.759,E2 -13915.759} C_VEL
LIN {X 0,Y 357.421,Z 333.257,A -85,B 0,C 180,E1 -13916.81,E2 -13916.81} C_VEL
LIN {X 0,Y 359.889,Z 343.711,A -85,B 0,C 180,E1 -13917.239,E2 -13917.239} C_VEL
LIN {X 0,Y 357.917,Z 422.992,A -85,B 0,C 180,E1 -13918.85,E2 -13918.85} C_VEL
LIN {X 0,Y 357.173,Z 436.474,A -85,B 0,C 180,E1 -13919.353,E2 -13919.353} C_VEL
LIN {X 0,Y 356.415,Z 449.223,A -85,B 0,C 180,E1 -13920.082,E2 -13920.082} C_VEL
LIN {X 0,Y 355.305,Z 461.214,A -85,B 0,C 180,E1 -13921.013,E2 -13921.013} C_VEL
LIN {X 0,Y 353.995,Z 472.912,A -85,B 0,C 180,E1 -13922.189,E2 -13922.189} C_VEL
LIN {X 0,Y 352.716,Z 482.735,A -85,B 0,C 180,E1 -13923.428,E2 -13923.428} C_VEL
LIN {X 0,Y 351.412,Z 491.848,A -85,B 0,C 180,E1 -13924.85,E2 -13924.85} C_VEL
LIN {X 0,Y 349.962,Z 501.013,A -85,B 0,C 180,E1 -13926.632,E2 -13926.632} C_VEL
LIN {X 0,Y 349.002,Z 507.622,A -85,B 0,C 180,E1 -13928.239,E2 -13928.239} C_VEL
LIN {X 0,Y 348.082,Z 513.243,A -85,B 0,C 180,E1 -13929.925,E2 -13929.925} C_VEL
LIN {X 0,Y 347.28,Z 518.611,A -85,B 0,C 180,E1 -13932.018,E2 -13932.018} C_VEL
LIN {X 0,Y 346.855,Z 521.523,A -85,B 0,C 180,E1 -13933.52,E2 -13933.52} C_VEL
LIN {X 0,Y 346.555,Z 523.3,A -85,B 0,C 180,E1 -13934.714,E2 -13934.714} C_VEL
LIN {X 0,Y 346.307,Z 525.449,A -85,B 0,C 180,E1 -13936.936,E2 -13936.936} C_VEL
LIN {X 0,Y 346.153,Z 526.083,A -85,B 0,C 180,E1 -13938.285,E2 -13938.285} C_VEL
LIN {X 0,Y 346.067,Z 525.854,A -85,B 0,C 180,E1 -13940.649,E2 -13940.649} C_VEL
LIN {X 0,Y 346.15,Z 525.154,A -85,B 0,C 180,E1 -13941.829,E2 -13941.829} C_VEL
LIN {X 0,Y 346.358,Z 522.973,A -85,B 0,C 180,E1 -13943.862,E2 -13943.862} C_VEL
LIN {X 0,Y 346.468,Z 519.402,A -85,B 0,C 180,E1 -13945.928,E2 -13945.928} C_VEL
LIN {X 0,Y 346.838,Z 515.246,A -85,B 0,C 180,E1 -13947.677,E2 -13947.677} C_VEL
LIN {X 0,Y 347.329,Z 508.928,A -85,B 0,C 180,E1 -13949.71,E2 -13949.71} C_VEL
LIN {X 0,Y 348.072,Z 502.041,A -85,B 0,C 180,E1 -13951.446,E2 -13951.446} C_VEL
LIN {X 0,Y 348.91,Z 493.427,A -85,B 0,C 180,E1 -13953.175,E2 -13953.175} C_VEL
LIN {X 0,Y 349.735,Z 484.616,A -85,B 0,C 180,E1 -13954.61,E2 -13954.61} C_VEL
LIN {X 0,Y 350.684,Z 474.929,A -85,B 0,C 180,E1 -13955.894,E2 -13955.894} C_VEL
LIN {X 0,Y 351.743,Z 465.686,A -85,B 0,C 180,E1 -13956.885,E2 -13956.885} C_VEL
LIN {X 0,Y 352.553,Z 454.334,A -85,B 0,C 180,E1 -13957.876,E2 -13957.876} C_VEL
LIN {X 0,Y 353.237,Z 441.349,A -85,B 0,C 180,E1 -13958.725,E2 -13958.725} C_VEL
LIN {X 0,Y 353.641,Z 429.199,A -85,B 0,C 180,E1 -13959.292,E2 -13959.292} C_VEL
LIN {X 0,Y 354.194,Z 417.035,A -85,B 0,C 180,E1 -13959.637,E2 -13959.637} C_VEL
LIN {X 0,Y 355.383,Z 340.651,A -85,B 0,C 180,E1 -13961.175,E2 -13961.175} C_VEL
LIN {X 0,Y 352.053,Z 323.083,A -85,B 0,C 180,E1 -13961.724,E2 -13961.724} C_VEL
LIN {X 0,Y 349.441,Z 315.049,A -85,B 0,C 180,E1 -13962.042,E2 -13962.042} C_VEL
LIN {X 0,Y 347.886,Z 307.153,A -85,B 0,C 180,E1 -13964.232,E2 -13964.232} C_VEL
LIN {X 0,Y 347.882,Z 307.153,A -85,B 0,C 180,E1 -13964.342,E2 -13964.342} C_VEL
LIN {X 0,Y 347.192,Z 307.234,A -85,B 0,C 180,E1 -13965.308,E2 -13965.308} C_VEL
LIN {X 0,Y 344.334,Z 307.591,A -85,B 0,C 180,E1 -13966.878,E2 -13966.878} C_VEL
LIN {X 0,Y 341.908,Z 307.895,A -85,B 0,C 180,E1 -13968.149,E2 -13968.149} C_VEL
LIN {X 0,Y 340.842,Z 308.026,A -85,B 0,C 180,E1 -13969.132,E2 -13969.132} C_VEL
LIN {X 0,Y 340.741,Z 308.037,A -85,B 0,C 180,E1 -13969.466,E2 -13969.466} C_VEL
LIN {X 0,Y 340.706,Z 308.043,A -85,B 0,C 180,E1 -13973.073,E2 -13973.073} C_VEL
LIN {X 0,Y 340.709,Z 308.041,A -85,B 0,C 180,E1 -13975.668,E2 -13975.668} C_VEL
LIN {X 0,Y 340.702,Z 308.042,A -85,B 0,C 180,E1 -13979.673,E2 -13979.673} C_VEL
LIN {X 0,Y 340.682,Z 308.047,A -85,B 0,C 180,E1 -13982.435,E2 -13982.435} C_VEL
LIN {X 0,Y 340.714,Z 308.043,A -85,B 0,C 180,E1 -13985.278,E2 -13985.278} C_VEL
LIN {X 0,Y 340.689,Z 308.044,A -85,B 0,C 180,E1 -13988.382,E2 -13988.382} C_VEL
LIN {X 0,Y 340.688,Z 308.043,A -85,B 0,C 180,E1 -13992.043,E2 -13992.043} C_VEL
LIN {X 0,Y 340.646,Z 308.049,A -85,B 0,C 180,E1 -13996.226,E2 -13996.226} C_VEL
LIN {X 0,Y 340.67,Z 308.047,A -85,B 0,C 180,E1 -13999.755,E2 -13999.755} C_VEL
LIN {X 0,Y 340.697,Z 308.048,A -85,B 0,C 180,E1 -14003.257,E2 -14003.257} C_VEL
LIN {X 0,Y 340.686,Z 308.044,A -85,B 0,C 180,E1 -14006.153,E2 -14006.153} C_VEL
LIN {X 0,Y 340.768,Z 308.033,A -85,B 0,C 180,E1 -14010.332,E2 -14010.332} C_VEL
LIN {X 0,Y 340.797,Z 308.031,A -85,B 0,C 180,E1 -14013.019,E2 -14013.019} C_VEL
LIN {X 0,Y 340.747,Z 308.043,A -85,B 0,C 180,E1 -14015.638,E2 -14015.638} C_VEL
LIN {X 0,Y 340.73,Z 308.041,A -85,B 0,C 180,E1 -14019.473,E2 -14019.473} C_VEL
LIN {X 0,Y 340.851,Z 308.028,A -85,B 0,C 180,E1 -14021.984,E2 -14021.984} C_VEL
LIN {X 0,Y 340.862,Z 308.026,A -85,B 0,C 180,E1 -14025.705,E2 -14025.705} C_VEL
LIN {X 0,Y 340.863,Z 308.021,A -85,B 0,C 180,E1 -14029.306,E2 -14029.306} C_VEL
LIN {X 0,Y 341.01,Z 308.004,A -85,B 0,C 180,E1 -14032.897,E2 -14032.897} C_VEL
LIN {X 0,Y 341.16,Z 307.986,A -85,B 0,C 180,E1 -14037.639,E2 -14037.639} C_VEL
LIN {X 0,Y 341.267,Z 307.974,A -85,B 0,C 180,E1 -14040,E2 -14040} C_VEL
LIN {X 0,Y 341.16,Z 307.99,A -85,B 0,C 180,E1 -14042.361,E2 -14042.361} C_VEL
LIN {X 0,Y 341.053,Z 307.999,A -85,B 0,C 180,E1 -14047.102,E2 -14047.102} C_VEL
LIN {X 0,Y 340.864,Z 308.026,A -85,B 0,C 180,E1 -14050.694,E2 -14050.694} C_VEL
LIN {X 0,Y 340.856,Z 308.025,A -85,B 0,C 180,E1 -14054.325,E2 -14054.325} C_VEL
LIN {X 0,Y 340.83,Z 308.029,A -85,B 0,C 180,E1 -14058.467,E2 -14058.467} C_VEL
LIN {X 0,Y 340.747,Z 308.036,A -85,B 0,C 180,E1 -14061.858,E2 -14061.858} C_VEL
LIN {X 0,Y 340.767,Z 308.034,A -85,B 0,C 180,E1 -14065.665,E2 -14065.665} C_VEL
LIN {X 0,Y 340.737,Z 308.038,A -85,B 0,C 180,E1 -14068.32,E2 -14068.32} C_VEL
LIN {X 0,Y 340.711,Z 308.046,A -85,B 0,C 180,E1 -14071.044,E2 -14071.044} C_VEL
LIN {X 0,Y 340.713,Z 308.047,A -85,B 0,C 180,E1 -14075.28,E2 -14075.28} C_VEL
LIN {X 0,Y 340.707,Z 308.041,A -85,B 0,C 180,E1 -14078.387,E2 -14078.387} C_VEL
LIN {X 0,Y 340.695,Z 308.044,A -85,B 0,C 180,E1 -14082.047,E2 -14082.047} C_VEL
LIN {X 0,Y 340.648,Z 308.049,A -85,B 0,C 180,E1 -14086.228,E2 -14086.228} C_VEL
LIN {X 0,Y 340.685,Z 308.049,A -85,B 0,C 180,E1 -14089.754,E2 -14089.754} C_VEL
LIN {X 0,Y 340.702,Z 308.044,A -85,B 0,C 180,E1 -14093.259,E2 -14093.259} C_VEL
LIN {X 0,Y 340.69,Z 308.047,A -85,B 0,C 180,E1 -14096.154,E2 -14096.154} C_VEL
LIN {X 0,Y 340.772,Z 308.195,A -85,B 0,C 180,E1 -14100.003,E2 -14100.003} C_VEL
LIN {X 0,Y 343.076,Z 319.192,A -85,B 0,C 180,E1 -14102.885,E2 -14102.885} C_VEL
LIN {X 0,Y 344.268,Z 326.032,A -85,B 0,C 180,E1 -14104.616,E2 -14104.616} C_VEL
LIN {X 0,Y 343.131,Z 338.82,A -85,B 0,C 180,E1 -14107.61,E2 -14107.61} C_VEL
LIN {X 0,Y 348.276,Z 376.11,A -85,B 0,C 180,E1 -14108.702,E2 -14108.702} C_VEL
LIN {X 0,Y 347.025,Z 448.194,A -85,B 0,C 180,E1 -14110.21,E2 -14110.21} C_VEL
LIN {X 0,Y 346.272,Z 461.991,A -85,B 0,C 180,E1 -14110.744,E2 -14110.744} C_VEL
LIN {X 0,Y 345.447,Z 474.394,A -85,B 0,C 180,E1 -14111.466,E2 -14111.466} C_VEL
LIN {X 0,Y 344.311,Z 487.078,A -85,B 0,C 180,E1 -14112.479,E2 -14112.479} C_VEL
LIN {X 0,Y 343.271,Z 498.388,A -85,B 0,C 180,E1 -14113.65,E2 -14113.65} C_VEL
LIN {X 0,Y 342.276,Z 509.214,A -85,B 0,C 180,E1 -14115.078,E2 -14115.078} C_VEL
LIN {X 0,Y 341.305,Z 518.546,A -85,B 0,C 180,E1 -14116.606,E2 -14116.606} C_VEL
LIN {X 0,Y 340.367,Z 527.322,A -85,B 0,C 180,E1 -14118.387,E2 -14118.387} C_VEL
LIN {X 0,Y 339.791,Z 534.318,A -85,B 0,C 180,E1 -14120.176,E2 -14120.176} C_VEL
LIN {X 0,Y 339.335,Z 540.729,A -85,B 0,C 180,E1 -14122.264,E2 -14122.264} C_VEL
LIN {X 0,Y 339.14,Z 545.028,A -85,B 0,C 180,E1 -14124.104,E2 -14124.104} C_VEL
LIN {X 0,Y 339.105,Z 547.134,A -85,B 0,C 180,E1 -14125.245,E2 -14125.245} C_VEL
LIN {X 0,Y 339.088,Z 548.855,A -85,B 0,C 180,E1 -14126.436,E2 -14126.436} C_VEL
LIN {X 0,Y 339.096,Z 551.076,A -85,B 0,C 180,E1 -14128.813,E2 -14128.813} C_VEL
LIN {X 0,Y 339.137,Z 551.578,A -85,B 0,C 180,E1 -14130.001,E2 -14130.001} C_VEL
LIN {X 0,Y 339.063,Z 551.646,A -85,B 0,C 180,E1 -14131.188,E2 -14131.188} C_VEL
LIN {X 0,Y 339.072,Z 550.628,A -85,B 0,C 180,E1 -14133.566,E2 -14133.566} C_VEL
LIN {X 0,Y 339.08,Z 549.529,A -85,B 0,C 180,E1 -14134.756,E2 -14134.756} C_VEL
LIN {X 0,Y 339.142,Z 547.983,A -85,B 0,C 180,E1 -14135.948,E2 -14135.948} C_VEL
LIN {X 0,Y 339.397,Z 544.891,A -85,B 0,C 180,E1 -14137.736,E2 -14137.736} C_VEL
LIN {X 0,Y 339.826,Z 540.758,A -85,B 0,C 180,E1 -14139.524,E2 -14139.524} C_VEL
LIN {X 0,Y 340.638,Z 534.463,A -85,B 0,C 180,E1 -14141.605,E2 -14141.605} C_VEL
LIN {X 0,Y 341.769,Z 527.634,A -85,B 0,C 180,E1 -14143.376,E2 -14143.376} C_VEL
LIN {X 0,Y 343.052,Z 519.149,A -85,B 0,C 180,E1 -14145.142,E2 -14145.142} C_VEL
LIN {X 0,Y 344.303,Z 510.45,A -85,B 0,C 180,E1 -14146.605,E2 -14146.605} C_VEL
LIN {X 0,Y 345.902,Z 499.765,A -85,B 0,C 180,E1 -14148.05,E2 -14148.05} C_VEL
LIN {X 0,Y 347.348,Z 489.144,A -85,B 0,C 180,E1 -14149.196,E2 -14149.196} C_VEL
LIN {X 0,Y 348.794,Z 477.278,A -85,B 0,C 180,E1 -14150.186,E2 -14150.186} C_VEL
LIN {X 0,Y 349.924,Z 464.973,A -85,B 0,C 180,E1 -14150.963,E2 -14150.963} C_VEL
LIN {X 0,Y 350.926,Z 452.322,A -85,B 0,C 180,E1 -14151.515,E2 -14151.515} C_VEL
LIN {X 0,Y 351.43,Z 437.415,A -85,B 0,C 180,E1 -14151.907,E2 -14151.907} C_VEL
LIN {X 0,Y 352.72,Z 376.934,A -85,B 0,C 180,E1 -14153.154,E2 -14153.154} C_VEL
LIN {X 0,Y 349.425,Z 357.515,A -85,B 0,C 180,E1 -14153.861,E2 -14153.861} C_VEL
LIN {X 0,Y 345.429,Z 338.175,A -85,B 0,C 180,E1 -14154.671,E2 -14154.671} C_VEL
LIN {X 0,Y 346.04,Z 333.099,A -85,B 0,C 180,E1 -14155.891,E2 -14155.891} C_VEL
LIN {X 0,Y 345.079,Z 326.668,A -85,B 0,C 180,E1 -14157.602,E2 -14157.602} C_VEL
LIN {X 0,Y 342.737,Z 316.234,A -85,B 0,C 180,E1 -14160.544,E2 -14160.544} C_VEL
LIN {X 0,Y 340.7,Z 308.042,A -85,B 0,C 180,E1 -14163.005,E2 -14163.005} C_VEL
LIN {X 0,Y 340.706,Z 308.045,A -85,B 0,C 180,E1 -14166.742,E2 -14166.742} C_VEL
LIN {X 0,Y 340.689,Z 308.047,A -85,B 0,C 180,E1 -14170.247,E2 -14170.247} C_VEL
LIN {X 0,Y 340.653,Z 308.052,A -85,B 0,C 180,E1 -14173.773,E2 -14173.773} C_VEL
LIN {X 0,Y 340.7,Z 308.043,A -85,B 0,C 180,E1 -14177.954,E2 -14177.954} C_VEL
LIN {X 0,Y 340.733,Z 308.039,A -85,B 0,C 180,E1 -14181.772,E2 -14181.772} C_VEL
LIN {X 0,Y 340.723,Z 308.036,A -85,B 0,C 180,E1 -14185.595,E2 -14185.595} C_VEL
LIN {X 0,Y 340.704,Z 308.042,A -85,B 0,C 180,E1 -14188.956,E2 -14188.956} C_VEL
LIN {X 0,Y 340.778,Z 308.034,A -85,B 0,C 180,E1 -14192.474,E2 -14192.474} C_VEL
LIN {X 0,Y 340.756,Z 308.038,A -85,B 0,C 180,E1 -14195.638,E2 -14195.638} C_VEL
LIN {X 0,Y 340.749,Z 308.04,A -85,B 0,C 180,E1 -14199.474,E2 -14199.474} C_VEL
LIN {X 0,Y 340.858,Z 308.022,A -85,B 0,C 180,E1 -14201.984,E2 -14201.984} C_VEL
LIN {X 0,Y 340.869,Z 308.017,A -85,B 0,C 180,E1 -14205.705,E2 -14205.705} C_VEL
LIN {X 0,Y 340.87,Z 308.018,A -85,B 0,C 180,E1 -14209.306,E2 -14209.306} C_VEL
LIN {X 0,Y 341.059,Z 307.994,A -85,B 0,C 180,E1 -14212.898,E2 -14212.898} C_VEL
LIN {X 0,Y 341.167,Z 307.984,A -85,B 0,C 180,E1 -14217.639,E2 -14217.639} C_VEL
LIN {X 0,Y 341.275,Z 307.965,A -85,B 0,C 180,E1 -14220,E2 -14220} C_VEL
LIN {X 0,Y 341.167,Z 307.979,A -85,B 0,C 180,E1 -14222.361,E2 -14222.361} C_VEL
LIN {X 0,Y 341.074,Z 307.99,A -85,B 0,C 180,E1 -14227.102,E2 -14227.102} C_VEL
LIN {X 0,Y 340.87,Z 308.021,A -85,B 0,C 180,E1 -14230.694,E2 -14230.694} C_VEL
LIN {X 0,Y 340.863,Z 308.026,A -85,B 0,C 180,E1 -14234.325,E2 -14234.325} C_VEL
LIN {X 0,Y 340.837,Z 308.03,A -85,B 0,C 180,E1 -14238.467,E2 -14238.467} C_VEL
LIN {X 0,Y 340.717,Z 308.039,A -85,B 0,C 180,E1 -14241.842,E2 -14241.842} C_VEL
LIN {X 0,Y 340.771,Z 308.033,A -85,B 0,C 180,E1 -14245.664,E2 -14245.664} C_VEL
LIN {X 0,Y 340.728,Z 308.034,A -85,B 0,C 180,E1 -14248.321,E2 -14248.321} C_VEL
LIN {X 0,Y 340.697,Z 308.041,A -85,B 0,C 180,E1 -14251.045,E2 -14251.045} C_VEL
LIN {X 0,Y 340.717,Z 308.04,A -85,B 0,C 180,E1 -14255.279,E2 -14255.279} C_VEL
LIN {X 0,Y 340.709,Z 308.042,A -85,B 0,C 180,E1 -14258.386,E2 -14258.386} C_VEL
LIN {X 0,Y 340.699,Z 308.044,A -85,B 0,C 180,E1 -14262.045,E2 -14262.045} C_VEL
LIN {X 0,Y 340.652,Z 308.051,A -85,B 0,C 180,E1 -14266.227,E2 -14266.227} C_VEL
LIN {X 0,Y 340.688,Z 308.048,A -85,B 0,C 180,E1 -14269.753,E2 -14269.753} C_VEL
LIN {X 0,Y 340.746,Z 308.144,A -85,B 0,C 180,E1 -14272.801,E2 -14272.801} C_VEL
LIN {X 0,Y 342.613,Z 315.777,A -85,B 0,C 180,E1 -14275.137,E2 -14275.137} C_VEL
LIN {X 0,Y 351.528,Z 336.244,A -85,B 0,C 180,E1 -14276.39,E2 -14276.39} C_VEL
LIN {X 0,Y 353.507,Z 344.681,A -85,B 0,C 180,E1 -14276.744,E2 -14276.744} C_VEL
LIN {X 0,Y 351.464,Z 423.605,A -85,B 0,C 180,E1 -14278.381,E2 -14278.381} C_VEL
LIN {X 0,Y 350.704,Z 436.965,A -85,B 0,C 180,E1 -14278.892,E2 -14278.892} C_VEL
LIN {X 0,Y 349.976,Z 448.6,A -85,B 0,C 180,E1 -14279.566,E2 -14279.566} C_VEL
LIN {X 0,Y 348.909,Z 459.948,A -85,B 0,C 180,E1 -14280.43,E2 -14280.43} C_VEL
LIN {X 0,Y 347.514,Z 471.926,A -85,B 0,C 180,E1 -14281.624,E2 -14281.624} C_VEL
LIN {X 0,Y 346.077,Z 482.621,A -85,B 0,C 180,E1 -14282.974,E2 -14282.974} C_VEL
LIN {X 0,Y 344.76,Z 491.444,A -85,B 0,C 180,E1 -14284.355,E2 -14284.355} C_VEL
LIN {X 0,Y 343.233,Z 500.622,A -85,B 0,C 180,E1 -14286.146,E2 -14286.146} C_VEL
LIN {X 0,Y 342.144,Z 507.697,A -85,B 0,C 180,E1 -14287.877,E2 -14287.877} C_VEL
LIN {X 0,Y 341.225,Z 513.074,A -85,B 0,C 180,E1 -14289.504,E2 -14289.504} C_VEL
LIN {X 0,Y 340.382,Z 518.032,A -85,B 0,C 180,E1 -14291.397,E2 -14291.397} C_VEL
LIN {X 0,Y 339.864,Z 521.535,A -85,B 0,C 180,E1 -14293.171,E2 -14293.171} C_VEL
LIN {X 0,Y 339.55,Z 523.392,A -85,B 0,C 180,E1 -14294.39,E2 -14294.39} C_VEL
LIN {X 0,Y 339.325,Z 524.765,A -85,B 0,C 180,E1 -14295.608,E2 -14295.608} C_VEL
LIN {X 0,Y 339.242,Z 525.73,A -85,B 0,C 180,E1 -14296.827,E2 -14296.827} C_VEL
LIN {X 0,Y 339.077,Z 526.303,A -85,B 0,C 180,E1 -14298.037,E2 -14298.037} C_VEL
LIN {X 0,Y 338.989,Z 526.451,A -85,B 0,C 180,E1 -14299.246,E2 -14299.246} C_VEL
LIN {X 0,Y 339.033,Z 525.516,A -85,B 0,C 180,E1 -14301.656,E2 -14301.656} C_VEL
LIN {X 0,Y 339.271,Z 523.215,A -85,B 0,C 180,E1 -14303.89,E2 -14303.89} C_VEL
LIN {X 0,Y 339.386,Z 519.958,A -85,B 0,C 180,E1 -14305.843,E2 -14305.843} C_VEL
LIN {X 0,Y 339.753,Z 515.888,A -85,B 0,C 180,E1 -14307.628,E2 -14307.628} C_VEL
LIN {X 0,Y 340.222,Z 509.667,A -85,B 0,C 180,E1 -14309.703,E2 -14309.703} C_VEL
LIN {X 0,Y 340.995,Z 502.884,A -85,B 0,C 180,E1 -14311.476,E2 -14311.476} C_VEL
LIN {X 0,Y 341.845,Z 494.454,A -85,B 0,C 180,E1 -14313.24,E2 -14313.24} C_VEL
LIN {X 0,Y 342.692,Z 485.793,A -85,B 0,C 180,E1 -14314.705,E2 -14314.705} C_VEL
LIN {X 0,Y 343.78,Z 475.125,A -85,B 0,C 180,E1 -14316.161,E2 -14316.161} C_VEL
LIN {X 0,Y 344.862,Z 465.869,A -85,B 0,C 180,E1 -14317.17,E2 -14317.17} C_VEL
LIN {X 0,Y 345.712,Z 454.49,A -85,B 0,C 180,E1 -14318.18,E2 -14318.18} C_VEL
LIN {X 0,Y 346.416,Z 441.467,A -85,B 0,C 180,E1 -14319.045,E2 -14319.045} C_VEL
LIN {X 0,Y 346.838,Z 429.261,A -85,B 0,C 180,E1 -14319.623,E2 -14319.623} C_VEL
LIN {X 0,Y 347.418,Z 416.954,A -85,B 0,C 180,E1 -14319.974,E2 -14319.974} C_VEL
LIN {X 0,Y 348.643,Z 341.545,A -85,B 0,C 180,E1 -14321.518,E2 -14321.518} C_VEL
LIN {X 0,Y 345.544,Z 325.188,A -85,B 0,C 180,E1 -14322.044,E2 -14322.044} C_VEL
LIN {X 0,Y 342.32,Z 315.301,A -85,B 0,C 180,E1 -14322.449,E2 -14322.449} C_VEL
LIN {X 0,Y 340.832,Z 308.029,A -85,B 0,C 180,E1 -14324.524,E2 -14324.524} C_VEL
LIN {X 0,Y 340.784,Z 308.038,A -85,B 0,C 180,E1 -14328.439,E2 -14328.439} C_VEL
LIN {X 0,Y 340.741,Z 308.037,A -85,B 0,C 180,E1 -14329.466,E2 -14329.466} C_VEL
LIN {X 0,Y 340.023,Z 308.133,A -85,B 0,C 180,E1 -14330.451,E2 -14330.451} C_VEL
LIN {X 0,Y 337.122,Z 308.49,A -85,B 0,C 180,E1 -14332.054,E2 -14332.054} C_VEL
LIN {X 0,Y 334.72,Z 308.787,A -85,B 0,C 180,E1 -14333.353,E2 -14333.353} C_VEL
LIN {X 0,Y 333.733,Z 308.914,A -85,B 0,C 180,E1 -14334.358,E2 -14334.358} C_VEL
LIN {X 0,Y 333.675,Z 308.918,A -85,B 0,C 180,E1 -14334.698,E2 -14334.698} C_VEL
LIN {X 0,Y 333.642,Z 308.921,A -85,B 0,C 180,E1 -14337.784,E2 -14337.784} C_VEL
LIN {X 0,Y 333.654,Z 308.922,A -85,B 0,C 180,E1 -14340.365,E2 -14340.365} C_VEL
LIN {X 0,Y 333.633,Z 308.925,A -85,B 0,C 180,E1 -14343.207,E2 -14343.207} C_VEL
LIN {X 0,Y 333.671,Z 308.918,A -85,B 0,C 180,E1 -14346.138,E2 -14346.138} C_VEL
LIN {X 0,Y 333.615,Z 308.928,A -85,B 0,C 180,E1 -14349.195,E2 -14349.195} C_VEL
LIN {X 0,Y 333.623,Z 308.925,A -85,B 0,C 180,E1 -14352.498,E2 -14352.498} C_VEL
LIN {X 0,Y 333.59,Z 308.928,A -85,B 0,C 180,E1 -14355.954,E2 -14355.954} C_VEL
LIN {X 0,Y 333.637,Z 308.926,A -85,B 0,C 180,E1 -14359.315,E2 -14359.315} C_VEL
LIN {X 0,Y 333.657,Z 308.923,A -85,B 0,C 180,E1 -14363.168,E2 -14363.168} C_VEL
LIN {X 0,Y 333.667,Z 308.924,A -85,B 0,C 180,E1 -14365.341,E2 -14365.341} C_VEL
LIN {X 0,Y 333.696,Z 308.917,A -85,B 0,C 180,E1 -14369.71,E2 -14369.71} C_VEL
LIN {X 0,Y 333.736,Z 308.909,A -85,B 0,C 180,E1 -14372.401,E2 -14372.401} C_VEL
LIN {X 0,Y 333.718,Z 308.913,A -85,B 0,C 180,E1 -14375.09,E2 -14375.09} C_VEL
LIN {X 0,Y 333.667,Z 308.917,A -85,B 0,C 180,E1 -14379.018,E2 -14379.018} C_VEL
LIN {X 0,Y 333.787,Z 308.906,A -85,B 0,C 180,E1 -14381.589,E2 -14381.589} C_VEL
LIN {X 0,Y 333.801,Z 308.904,A -85,B 0,C 180,E1 -14385.576,E2 -14385.576} C_VEL
LIN {X 0,Y 333.826,Z 308.897,A -85,B 0,C 180,E1 -14389.078,E2 -14389.078} C_VEL
LIN {X 0,Y 333.962,Z 308.882,A -85,B 0,C 180,E1 -14392.746,E2 -14392.746} C_VEL
LIN {X 0,Y 333.798,Z 308.902,A -85,B 0,C 180,E1 -14395.169,E2 -14395.169} C_VEL
LIN {X 0,Y 334.097,Z 308.865,A -85,B 0,C 180,E1 -14397.589,E2 -14397.589} C_VEL
LIN {X 0,Y 334.219,Z 308.851,A -85,B 0,C 180,E1 -14400,E2 -14400} C_VEL
LIN {X 0,Y 334.097,Z 308.87,A -85,B 0,C 180,E1 -14402.411,E2 -14402.411} C_VEL
LIN {X 0,Y 334.008,Z 308.878,A -85,B 0,C 180,E1 -14406.039,E2 -14406.039} C_VEL
LIN {X 0,Y 333.977,Z 308.885,A -85,B 0,C 180,E1 -14408.502,E2 -14408.502} C_VEL
LIN {X 0,Y 333.784,Z 308.904,A -85,B 0,C 180,E1 -14412.155,E2 -14412.155} C_VEL
LIN {X 0,Y 333.771,Z 308.905,A -85,B 0,C 180,E1 -14415.887,E2 -14415.887} C_VEL
LIN {X 0,Y 333.789,Z 308.907,A -85,B 0,C 180,E1 -14418.655,E2 -14418.655} C_VEL
LIN {X 0,Y 333.686,Z 308.917,A -85,B 0,C 180,E1 -14422.279,E2 -14422.279} C_VEL
LIN {X 0,Y 333.73,Z 308.911,A -85,B 0,C 180,E1 -14426.247,E2 -14426.247} C_VEL
LIN {X 0,Y 333.706,Z 308.919,A -85,B 0,C 180,E1 -14428.973,E2 -14428.973} C_VEL
LIN {X 0,Y 333.646,Z 308.922,A -85,B 0,C 180,E1 -14432.59,E2 -14432.59} C_VEL
LIN {X 0,Y 333.672,Z 308.918,A -85,B 0,C 180,E1 -14436.14,E2 -14436.14} C_VEL
LIN {X 0,Y 333.643,Z 308.926,A -85,B 0,C 180,E1 -14439.193,E2 -14439.193} C_VEL
LIN {X 0,Y 333.629,Z 308.923,A -85,B 0,C 180,E1 -14442.501,E2 -14442.501} C_VEL
LIN {X 0,Y 333.593,Z 308.93,A -85,B 0,C 180,E1 -14445.956,E2 -14445.956} C_VEL
LIN {X 0,Y 333.644,Z 308.924,A -85,B 0,C 180,E1 -14449.316,E2 -14449.316} C_VEL
LIN {X 0,Y 333.662,Z 308.92,A -85,B 0,C 180,E1 -14453.169,E2 -14453.169} C_VEL
LIN {X 0,Y 333.672,Z 308.921,A -85,B 0,C 180,E1 -14455.342,E2 -14455.342} C_VEL
LIN {X 0,Y 333.734,Z 309.089,A -85,B 0,C 180,E1 -14459.702,E2 -14459.702} C_VEL
LIN {X 0,Y 335.998,Z 319.915,A -85,B 0,C 180,E1 -14462.603,E2 -14462.603} C_VEL
LIN {X 0,Y 337.319,Z 328.115,A -85,B 0,C 180,E1 -14464.716,E2 -14464.716} C_VEL
LIN {X 0,Y 336.23,Z 338.564,A -85,B 0,C 180,E1 -14467.208,E2 -14467.208} C_VEL
LIN {X 0,Y 341.524,Z 377.22,A -85,B 0,C 180,E1 -14468.364,E2 -14468.364} C_VEL
LIN {X 0,Y 340.246,Z 446.963,A -85,B 0,C 180,E1 -14469.838,E2 -14469.838} C_VEL
LIN {X 0,Y 339.516,Z 460.314,A -85,B 0,C 180,E1 -14470.345,E2 -14470.345} C_VEL
LIN {X 0,Y 338.661,Z 473.129,A -85,B 0,C 180,E1 -14471.08,E2 -14471.08} C_VEL
LIN {X 0,Y 337.711,Z 484.494,A -85,B 0,C 180,E1 -14471.968,E2 -14471.968} C_VEL
LIN {X 0,Y 336.552,Z 496.222,A -85,B 0,C 180,E1 -14473.158,E2 -14473.158} C_VEL
LIN {X 0,Y 335.436,Z 507.397,A -85,B 0,C 180,E1 -14474.597,E2 -14474.597} C_VEL
LIN {X 0,Y 334.504,Z 516.255,A -85,B 0,C 180,E1 -14476.019,E2 -14476.019} C_VEL
LIN {X 0,Y 333.561,Z 525.394,A -85,B 0,C 180,E1 -14477.838,E2 -14477.838} C_VEL
LIN {X 0,Y 332.829,Z 532.748,A -85,B 0,C 180,E1 -14479.661,E2 -14479.661} C_VEL
LIN {X 0,Y 332.374,Z 538.631,A -85,B 0,C 180,E1 -14481.489,E2 -14481.489} C_VEL
LIN {X 0,Y 332.115,Z 543.252,A -85,B 0,C 180,E1 -14483.317,E2 -14483.317} C_VEL
LIN {X 0,Y 332.009,Z 546.756,A -85,B 0,C 180,E1 -14485.144,E2 -14485.144} C_VEL
LIN {X 0,Y 332.014,Z 548.508,A -85,B 0,C 180,E1 -14486.36,E2 -14486.36} C_VEL
LIN {X 0,Y 331.998,Z 550.765,A -85,B 0,C 180,E1 -14488.788,E2 -14488.788} C_VEL
LIN {X 0,Y 332.042,Z 551.298,A -85,B 0,C 180,E1 -14490.001,E2 -14490.001} C_VEL
LIN {X 0,Y 331.965,Z 551.39,A -85,B 0,C 180,E1 -14491.214,E2 -14491.214} C_VEL
LIN {X 0,Y 331.997,Z 550.409,A -85,B 0,C 180,E1 -14493.642,E2 -14493.642} C_VEL
LIN {X 0,Y 332.037,Z 548.165,A -85,B 0,C 180,E1 -14495.833,E2 -14495.833} C_VEL
LIN {X 0,Y 332.335,Z 544.766,A -85,B 0,C 180,E1 -14497.901,E2 -14497.901} C_VEL
LIN {X 0,Y 332.801,Z 540.675,A -85,B 0,C 180,E1 -14499.727,E2 -14499.727} C_VEL
LIN {X 0,Y 333.657,Z 534.426,A -85,B 0,C 180,E1 -14501.852,E2 -14501.852} C_VEL
LIN {X 0,Y 334.842,Z 527.65,A -85,B 0,C 180,E1 -14503.658,E2 -14503.658} C_VEL
LIN {X 0,Y 336.178,Z 519.259,A -85,B 0,C 180,E1 -14505.459,E2 -14505.459} C_VEL
LIN {X 0,Y 337.511,Z 510.642,A -85,B 0,C 180,E1 -14506.95,E2 -14506.95} C_VEL
LIN {X 0,Y 339.159,Z 500.055,A -85,B 0,C 180,E1 -14508.422,E2 -14508.422} C_VEL
LIN {X 0,Y 340.686,Z 489.565,A -85,B 0,C 180,E1 -14509.586,E2 -14509.586} C_VEL
LIN {X 0,Y 342.186,Z 477.96,A -85,B 0,C 180,E1 -14510.593,E2 -14510.593} C_VEL
LIN {X 0,Y 343.354,Z 465.947,A -85,B 0,C 180,E1 -14511.383,E2 -14511.383} C_VEL
LIN {X 0,Y 344.434,Z 452.899,A -85,B 0,C 180,E1 -14511.981,E2 -14511.981} C_VEL
LIN {X 0,Y 344.966,Z 440.517,A -85,B 0,C 180,E1 -14512.339,E2 -14512.339} C_VEL
LIN {X 0,Y 346.381,Z 378.002,A -85,B 0,C 180,E1 -14513.649,E2 -14513.649} C_VEL
LIN {X 0,Y 343.033,Z 358.318,A -85,B 0,C 180,E1 -14514.388,E2 -14514.388} C_VEL
LIN {X 0,Y 338.753,Z 337.903,A -85,B 0,C 180,E1 -14515.273,E2 -14515.273} C_VEL
LIN {X 0,Y 339.135,Z 333.52,A -85,B 0,C 180,E1 -14516.364,E2 -14516.364} C_VEL
LIN {X 0,Y 337.364,Z 324.204,A -85,B 0,C 180,E1 -14518.961,E2 -14518.961} C_VEL
LIN {X 0,Y 334.755,Z 313.327,A -85,B 0,C 180,E1 -14522.178,E2 -14522.178} C_VEL
LIN {X 0,Y 333.663,Z 308.92,A -85,B 0,C 180,E1 -14523.567,E2 -14523.567} C_VEL
LIN {X 0,Y 333.667,Z 308.922,A -85,B 0,C 180,E1 -14526.832,E2 -14526.832} C_VEL
LIN {X 0,Y 333.648,Z 308.925,A -85,B 0,C 180,E1 -14530.767,E2 -14530.767} C_VEL
LIN {X 0,Y 333.595,Z 308.931,A -85,B 0,C 180,E1 -14534.25,E2 -14534.25} C_VEL
LIN {X 0,Y 333.643,Z 308.922,A -85,B 0,C 180,E1 -14537.618,E2 -14537.618} C_VEL
LIN {X 0,Y 333.653,Z 308.923,A -85,B 0,C 180,E1 -14541.202,E2 -14541.202} C_VEL
LIN {X 0,Y 333.677,Z 308.917,A -85,B 0,C 180,E1 -14543.861,E2 -14543.861} C_VEL
LIN {X 0,Y 333.644,Z 308.924,A -85,B 0,C 180,E1 -14547.413,E2 -14547.413} C_VEL
LIN {X 0,Y 333.711,Z 308.916,A -85,B 0,C 180,E1 -14551.028,E2 -14551.028} C_VEL
LIN {X 0,Y 333.736,Z 308.91,A -85,B 0,C 180,E1 -14553.754,E2 -14553.754} C_VEL
LIN {X 0,Y 333.72,Z 308.912,A -85,B 0,C 180,E1 -14557.914,E2 -14557.914} C_VEL
LIN {X 0,Y 333.795,Z 308.9,A -85,B 0,C 180,E1 -14561.589,E2 -14561.589} C_VEL
LIN {X 0,Y 333.808,Z 308.896,A -85,B 0,C 180,E1 -14565.576,E2 -14565.576} C_VEL
LIN {X 0,Y 333.833,Z 308.896,A -85,B 0,C 180,E1 -14569.078,E2 -14569.078} C_VEL
LIN {X 0,Y 334.006,Z 308.873,A -85,B 0,C 180,E1 -14572.747,E2 -14572.747} C_VEL
LIN {X 0,Y 333.808,Z 308.892,A -85,B 0,C 180,E1 -14575.169,E2 -14575.169} C_VEL
LIN {X 0,Y 334.104,Z 308.863,A -85,B 0,C 180,E1 -14577.589,E2 -14577.589} C_VEL
LIN {X 0,Y 334.226,Z 308.843,A -85,B 0,C 180,E1 -14580,E2 -14580} C_VEL
LIN {X 0,Y 334.104,Z 308.858,A -85,B 0,C 180,E1 -14582.411,E2 -14582.411} C_VEL
LIN {X 0,Y 334.023,Z 308.868,A -85,B 0,C 180,E1 -14587.252,E2 -14587.252} C_VEL
LIN {X 0,Y 333.833,Z 308.896,A -85,B 0,C 180,E1 -14590.922,E2 -14590.922} C_VEL
LIN {X 0,Y 333.808,Z 308.905,A -85,B 0,C 180,E1 -14594.634,E2 -14594.634} C_VEL
LIN {X 0,Y 333.796,Z 308.908,A -85,B 0,C 180,E1 -14598.655,E2 -14598.655} C_VEL
LIN {X 0,Y 333.656,Z 308.921,A -85,B 0,C 180,E1 -14602.281,E2 -14602.281} C_VEL
LIN {X 0,Y 333.734,Z 308.91,A -85,B 0,C 180,E1 -14606.246,E2 -14606.246} C_VEL
LIN {X 0,Y 333.69,Z 308.914,A -85,B 0,C 180,E1 -14608.974,E2 -14608.974} C_VEL
LIN {X 0,Y 333.643,Z 308.919,A -85,B 0,C 180,E1 -14612.587,E2 -14612.587} C_VEL
LIN {X 0,Y 333.676,Z 308.918,A -85,B 0,C 180,E1 -14616.139,E2 -14616.139} C_VEL
LIN {X 0,Y 333.646,Z 308.926,A -85,B 0,C 180,E1 -14619.192,E2 -14619.192} C_VEL
LIN {X 0,Y 333.632,Z 308.924,A -85,B 0,C 180,E1 -14622.5,E2 -14622.5} C_VEL
LIN {X 0,Y 333.596,Z 308.931,A -85,B 0,C 180,E1 -14625.955,E2 -14625.955} C_VEL
LIN {X 0,Y 333.647,Z 308.926,A -85,B 0,C 180,E1 -14629.315,E2 -14629.315} C_VEL
LIN {X 0,Y 333.71,Z 309.058,A -85,B 0,C 180,E1 -14632.261,E2 -14632.261} C_VEL
LIN {X 0,Y 335.468,Z 316.106,A -85,B 0,C 180,E1 -14634.474,E2 -14634.474} C_VEL
LIN {X 0,Y 344.876,Z 337.255,A -85,B 0,C 180,E1 -14635.841,E2 -14635.841} C_VEL
LIN {X 0,Y 346.581,Z 342.917,A -85,B 0,C 180,E1 -14636.12,E2 -14636.12} C_VEL
LIN {X 0,Y 347.148,Z 345.718,A -85,B 0,C 180,E1 -14636.233,E2 -14636.233} C_VEL
LIN {X 0,Y 345.066,Z 423.718,A -85,B 0,C 180,E1 -14637.878,E2 -14637.878} C_VEL
LIN {X 0,Y 344.248,Z 437.467,A -85,B 0,C 180,E1 -14638.413,E2 -14638.413} C_VEL
LIN {X 0,Y 343.434,Z 449.735,A -85,B 0,C 180,E1 -14639.144,E2 -14639.144} C_VEL
LIN {X 0,Y 342.304,Z 460.983,A -85,B 0,C 180,E1 -14640.036,E2 -14640.036} C_VEL
LIN {X 0,Y 340.914,Z 472.294,A -85,B 0,C 180,E1 -14641.192,E2 -14641.192} C_VEL
LIN {X 0,Y 339.41,Z 482.971,A -85,B 0,C 180,E1 -14642.566,E2 -14642.566} C_VEL
LIN {X 0,Y 337.892,Z 492.481,A -85,B 0,C 180,E1 -14644.1,E2 -14644.1} C_VEL
LIN {X 0,Y 336.319,Z 501.627,A -85,B 0,C 180,E1 -14645.953,E2 -14645.953} C_VEL
LIN {X 0,Y 335.114,Z 508.936,A -85,B 0,C 180,E1 -14647.821,E2 -14647.821} C_VEL
LIN {X 0,Y 334.059,Z 514.696,A -85,B 0,C 180,E1 -14649.688,E2 -14649.688} C_VEL
LIN {X 0,Y 333.248,Z 519.325,A -85,B 0,C 180,E1 -14651.626,E2 -14651.626} C_VEL
LIN {X 0,Y 332.892,Z 521.546,A -85,B 0,C 180,E1 -14652.808,E2 -14652.808} C_VEL
LIN {X 0,Y 332.535,Z 523.459,A -85,B 0,C 180,E1 -14654.052,E2 -14654.052} C_VEL
LIN {X 0,Y 332.299,Z 524.899,A -85,B 0,C 180,E1 -14655.297,E2 -14655.297} C_VEL
LIN {X 0,Y 332.173,Z 526.014,A -85,B 0,C 180,E1 -14656.718,E2 -14656.718} C_VEL
LIN {X 0,Y 331.914,Z 526.728,A -85,B 0,C 180,E1 -14659.014,E2 -14659.014} C_VEL
LIN {X 0,Y 331.872,Z 526.502,A -85,B 0,C 180,E1 -14660.246,E2 -14660.246} C_VEL
LIN {X 0,Y 331.936,Z 525.877,A -85,B 0,C 180,E1 -14661.476,E2 -14661.476} C_VEL
LIN {X 0,Y 332.019,Z 524.866,A -85,B 0,C 180,E1 -14662.703,E2 -14662.703} C_VEL
LIN {X 0,Y 332.18,Z 523.446,A -85,B 0,C 180,E1 -14663.927,E2 -14663.927} C_VEL
LIN {X 0,Y 332.307,Z 520.503,A -85,B 0,C 180,E1 -14665.754,E2 -14665.754} C_VEL
LIN {X 0,Y 332.666,Z 516.519,A -85,B 0,C 180,E1 -14667.578,E2 -14667.578} C_VEL
LIN {X 0,Y 333.125,Z 510.405,A -85,B 0,C 180,E1 -14669.697,E2 -14669.697} C_VEL
LIN {X 0,Y 333.918,Z 503.726,A -85,B 0,C 180,E1 -14671.507,E2 -14671.507} C_VEL
LIN {X 0,Y 334.786,Z 495.463,A -85,B 0,C 180,E1 -14673.309,E2 -14673.309} C_VEL
LIN {X 0,Y 335.673,Z 486.967,A -85,B 0,C 180,E1 -14674.803,E2 -14674.803} C_VEL
LIN {X 0,Y 336.748,Z 476.491,A -85,B 0,C 180,E1 -14676.29,E2 -14676.29} C_VEL
LIN {X 0,Y 337.745,Z 467.493,A -85,B 0,C 180,E1 -14677.322,E2 -14677.322} C_VEL
LIN {X 0,Y 338.653,Z 458.154,A -85,B 0,C 180,E1 -14678.202,E2 -14678.202} C_VEL
LIN {X 0,Y 339.44,Z 445.276,A -85,B 0,C 180,E1 -14679.158,E2 -14679.158} C_VEL
LIN {X 0,Y 339.895,Z 432.922,A -85,B 0,C 180,E1 -14679.821,E2 -14679.821} C_VEL
LIN {X 0,Y 340.543,Z 419.836,A -85,B 0,C 180,E1 -14680.252,E2 -14680.252} C_VEL
LIN {X 0,Y 342.006,Z 342.995,A -85,B 0,C 180,E1 -14681.858,E2 -14681.858} C_VEL
LIN {X 0,Y 339.054,Z 327.29,A -85,B 0,C 180,E1 -14682.373,E2 -14682.373} C_VEL
LIN {X 0,Y 335.127,Z 315.444,A -85,B 0,C 180,E1 -14682.906,E2 -14682.906} C_VEL
LIN {X 0,Y 333.785,Z 308.905,A -85,B 0,C 180,E1 -14684.79,E2 -14684.79} C_VEL
LIN {X 0,Y 333.751,Z 308.912,A -85,B 0,C 180,E1 -14688.632,E2 -14688.632} C_VEL
LIN {X 0,Y 333.65,Z 308.925,A -85,B 0,C 180,E1 -14692.28,E2 -14692.28} C_VEL
LIN {X 0,Y 333.675,Z 308.918,A -85,B 0,C 180,E1 -14694.698,E2 -14694.698} C_VEL
LIN {X 0,Y 333.061,Z 308.999,A -85,B 0,C 180,E1 -14695.706,E2 -14695.706} C_VEL
LIN {X 0,Y 330.206,Z 309.353,A -85,B 0,C 180,E1 -14697.345,E2 -14697.345} C_VEL
LIN {X 0,Y 327.747,Z 309.661,A -85,B 0,C 180,E1 -14698.673,E2 -14698.673} C_VEL
LIN {X 0,Y 326.686,Z 309.788,A -85,B 0,C 180,E1 -14699.701,E2 -14699.701} C_VEL
LIN {X 0,Y 326.599,Z 309.799,A -85,B 0,C 180,E1 -14700.05,E2 -14700.05} C_VEL
LIN {X 0,Y 326.603,Z 309.799,A -85,B 0,C 180,E1 -14704.018,E2 -14704.018} C_VEL
LIN {X 0,Y 326.619,Z 309.798,A -85,B 0,C 180,E1 -14707.237,E2 -14707.237} C_VEL
LIN {X 0,Y 326.539,Z 309.811,A -85,B 0,C 180,E1 -14711.124,E2 -14711.124} C_VEL
LIN {X 0,Y 326.555,Z 309.804,A -85,B 0,C 180,E1 -14713.525,E2 -14713.525} C_VEL
LIN {X 0,Y 326.57,Z 309.807,A -85,B 0,C 180,E1 -14717.027,E2 -14717.027} C_VEL
LIN {X 0,Y 326.593,Z 309.8,A -85,B 0,C 180,E1 -14720.775,E2 -14720.775} C_VEL
LIN {X 0,Y 326.605,Z 309.798,A -85,B 0,C 180,E1 -14724.48,E2 -14724.48} C_VEL
LIN {X 0,Y 326.601,Z 309.803,A -85,B 0,C 180,E1 -14727.455,E2 -14727.455} C_VEL
LIN {X 0,Y 326.654,Z 309.79,A -85,B 0,C 180,E1 -14730.34,E2 -14730.34} C_VEL
LIN {X 0,Y 326.683,Z 309.788,A -85,B 0,C 180,E1 -14734.516,E2 -14734.516} C_VEL
LIN {X 0,Y 326.613,Z 309.795,A -85,B 0,C 180,E1 -14738.543,E2 -14738.543} C_VEL
LIN {X 0,Y 326.737,Z 309.78,A -85,B 0,C 180,E1 -14741.177,E2 -14741.177} C_VEL
LIN {X 0,Y 326.756,Z 309.781,A -85,B 0,C 180,E1 -14745.433,E2 -14745.433} C_VEL
LIN {X 0,Y 326.762,Z 309.776,A -85,B 0,C 180,E1 -14748.839,E2 -14748.839} C_VEL
LIN {X 0,Y 326.916,Z 309.76,A -85,B 0,C 180,E1 -14752.589,E2 -14752.589} C_VEL
LIN {X 0,Y 326.764,Z 309.778,A -85,B 0,C 180,E1 -14755.065,E2 -14755.065} C_VEL
LIN {X 0,Y 327.038,Z 309.744,A -85,B 0,C 180,E1 -14757.537,E2 -14757.537} C_VEL
LIN {X 0,Y 327.171,Z 309.729,A -85,B 0,C 180,E1 -14760,E2 -14760} C_VEL
LIN {X 0,Y 327.038,Z 309.749,A -85,B 0,C 180,E1 -14762.463,E2 -14762.463} C_VEL
LIN {X 0,Y 326.983,Z 309.754,A -85,B 0,C 180,E1 -14766.17,E2 -14766.17} C_VEL
LIN {X 0,Y 326.907,Z 309.764,A -85,B 0,C 180,E1 -14768.655,E2 -14768.655} C_VEL
LIN {X 0,Y 326.728,Z 309.784,A -85,B 0,C 180,E1 -14772.422,E2 -14772.422} C_VEL
LIN {X 0,Y 326.747,Z 309.784,A -85,B 0,C 180,E1 -14774.958,E2 -14774.958} C_VEL
LIN {X 0,Y 326.726,Z 309.789,A -85,B 0,C 180,E1 -14778.839,E2 -14778.839} C_VEL
LIN {X 0,Y 326.614,Z 309.801,A -85,B 0,C 180,E1 -14782.788,E2 -14782.788} C_VEL
LIN {X 0,Y 326.684,Z 309.79,A -85,B 0,C 180,E1 -14785.484,E2 -14785.484} C_VEL
LIN {X 0,Y 326.656,Z 309.793,A -85,B 0,C 180,E1 -14789.66,E2 -14789.66} C_VEL
LIN {X 0,Y 326.618,Z 309.801,A -85,B 0,C 180,E1 -14792.949,E2 -14792.949} C_VEL
LIN {X 0,Y 326.608,Z 309.802,A -85,B 0,C 180,E1 -14795.52,E2 -14795.52} C_VEL
LIN {X 0,Y 326.607,Z 309.803,A -85,B 0,C 180,E1 -14799.228,E2 -14799.228} C_VEL
LIN {X 0,Y 326.572,Z 309.805,A -85,B 0,C 180,E1 -14802.973,E2 -14802.973} C_VEL
LIN {X 0,Y 326.573,Z 309.804,A -85,B 0,C 180,E1 -14807.029,E2 -14807.029} C_VEL
LIN {X 0,Y 326.608,Z 309.798,A -85,B 0,C 180,E1 -14810.774,E2 -14810.774} C_VEL
LIN {X 0,Y 326.61,Z 309.799,A -85,B 0,C 180,E1 -14814.481,E2 -14814.481} C_VEL
LIN {X 0,Y 326.606,Z 309.802,A -85,B 0,C 180,E1 -14817.457,E2 -14817.457} C_VEL
LIN {X 0,Y 326.657,Z 309.983,A -85,B 0,C 180,E1 -14819.384,E2 -14819.384} C_VEL
LIN {X 0,Y 328.927,Z 320.621,A -85,B 0,C 180,E1 -14822.309,E2 -14822.309} C_VEL
LIN {X 0,Y 330.332,Z 328.844,A -85,B 0,C 180,E1 -14824.481,E2 -14824.481} C_VEL
LIN {X 0,Y 329.363,Z 338.311,A -85,B 0,C 180,E1 -14826.789,E2 -14826.789} C_VEL
LIN {X 0,Y 334.749,Z 377.544,A -85,B 0,C 180,E1 -14827.994,E2 -14827.994} C_VEL
LIN {X 0,Y 333.464,Z 446.795,A -85,B 0,C 180,E1 -14829.49,E2 -14829.49} C_VEL
LIN {X 0,Y 332.713,Z 460.116,A -85,B 0,C 180,E1 -14830.006,E2 -14830.006} C_VEL
LIN {X 0,Y 331.825,Z 472.917,A -85,B 0,C 180,E1 -14830.756,E2 -14830.756} C_VEL
LIN {X 0,Y 330.763,Z 485.069,A -85,B 0,C 180,E1 -14831.736,E2 -14831.736} C_VEL
LIN {X 0,Y 329.575,Z 496.646,A -85,B 0,C 180,E1 -14832.951,E2 -14832.951} C_VEL
LIN {X 0,Y 328.553,Z 506.712,A -85,B 0,C 180,E1 -14834.278,E2 -14834.278} C_VEL
LIN {X 0,Y 327.59,Z 515.6,A -85,B 0,C 180,E1 -14835.718,E2 -14835.718} C_VEL
LIN {X 0,Y 326.57,Z 524.813,A -85,B 0,C 180,E1 -14837.573,E2 -14837.573} C_VEL
LIN {X 0,Y 325.812,Z 532.225,A -85,B 0,C 180,E1 -14839.436,E2 -14839.436} C_VEL
LIN {X 0,Y 325.326,Z 538.161,A -85,B 0,C 180,E1 -14841.303,E2 -14841.303} C_VEL
LIN {X 0,Y 325.048,Z 542.83,A -85,B 0,C 180,E1 -14843.171,E2 -14843.171} C_VEL
LIN {X 0,Y 324.917,Z 546.371,A -85,B 0,C 180,E1 -14845.037,E2 -14845.037} C_VEL
LIN {X 0,Y 324.94,Z 548.161,A -85,B 0,C 180,E1 -14846.28,E2 -14846.28} C_VEL
LIN {X 0,Y 324.903,Z 550.455,A -85,B 0,C 180,E1 -14848.761,E2 -14848.761} C_VEL
LIN {X 0,Y 324.947,Z 551.011,A -85,B 0,C 180,E1 -14850.001,E2 -14850.001} C_VEL
LIN {X 0,Y 324.871,Z 551.134,A -85,B 0,C 180,E1 -14851.24,E2 -14851.24} C_VEL
LIN {X 0,Y 324.901,Z 550.189,A -85,B 0,C 180,E1 -14853.721,E2 -14853.721} C_VEL
LIN {X 0,Y 324.949,Z 548.183,A -85,B 0,C 180,E1 -14855.793,E2 -14855.793} C_VEL
LIN {X 0,Y 325.266,Z 544.642,A -85,B 0,C 180,E1 -14858.074,E2 -14858.074} C_VEL
LIN {X 0,Y 325.79,Z 540.595,A -85,B 0,C 180,E1 -14859.938,E2 -14859.938} C_VEL
LIN {X 0,Y 326.691,Z 534.4,A -85,B 0,C 180,E1 -14862.108,E2 -14862.108} C_VEL
LIN {X 0,Y 327.933,Z 527.679,A -85,B 0,C 180,E1 -14863.952,E2 -14863.952} C_VEL
LIN {X 0,Y 329.31,Z 519.367,A -85,B 0,C 180,E1 -14865.79,E2 -14865.79} C_VEL
LIN {X 0,Y 330.731,Z 510.843,A -85,B 0,C 180,E1 -14867.308,E2 -14867.308} C_VEL
LIN {X 0,Y 332.434,Z 500.352,A -85,B 0,C 180,E1 -14868.809,E2 -14868.809} C_VEL
LIN {X 0,Y 334.038,Z 489.98,A -85,B 0,C 180,E1 -14869.993,E2 -14869.993} C_VEL
LIN {X 0,Y 335.596,Z 478.609,A -85,B 0,C 180,E1 -14871.016,E2 -14871.016} C_VEL
LIN {X 0,Y 336.821,Z 466.918,A -85,B 0,C 180,E1 -14871.819,E2 -14871.819} C_VEL
LIN {X 0,Y 337.963,Z 453.471,A -85,B 0,C 180,E1 -14872.465,E2 -14872.465} C_VEL
LIN {X 0,Y 338.591,Z 440.115,A -85,B 0,C 180,E1 -14872.864,E2 -14872.864} C_VEL
LIN {X 0,Y 340.077,Z 379.248,A -85,B 0,C 180,E1 -14874.157,E2 -14874.157} C_VEL
LIN {X 0,Y 336.976,Z 360.721,A -85,B 0,C 180,E1 -14874.871,E2 -14874.871} C_VEL
LIN {X 0,Y 332.568,Z 339.811,A -85,B 0,C 180,E1 -14875.786,E2 -14875.786} C_VEL
LIN {X 0,Y 332.155,Z 337.668,A -85,B 0,C 180,E1 -14875.888,E2 -14875.888} C_VEL
LIN {X 0,Y 332.232,Z 334.677,A -85,B 0,C 180,E1 -14876.667,E2 -14876.667} C_VEL
LIN {X 0,Y 330.179,Z 324.24,A -85,B 0,C 180,E1 -14879.662,E2 -14879.662} C_VEL
LIN {X 0,Y 327.362,Z 312.895,A -85,B 0,C 180,E1 -14883.146,E2 -14883.146} C_VEL
LIN {X 0,Y 326.633,Z 309.802,A -85,B 0,C 180,E1 -14884.203,E2 -14884.203} C_VEL
LIN {X 0,Y 326.629,Z 309.8,A -85,B 0,C 180,E1 -14887.238,E2 -14887.238} C_VEL
LIN {X 0,Y 326.579,Z 309.806,A -85,B 0,C 180,E1 -14891.131,E2 -14891.131} C_VEL
LIN {X 0,Y 326.529,Z 309.81,A -85,B 0,C 180,E1 -14894.743,E2 -14894.743} C_VEL
LIN {X 0,Y 326.577,Z 309.804,A -85,B 0,C 180,E1 -14898.154,E2 -14898.154} C_VEL
LIN {X 0,Y 326.598,Z 309.801,A -85,B 0,C 180,E1 -14901.388,E2 -14901.388} C_VEL
LIN {X 0,Y 326.62,Z 309.799,A -85,B 0,C 180,E1 -14904.851,E2 -14904.851} C_VEL
LIN {X 0,Y 326.608,Z 309.801,A -85,B 0,C 180,E1 -14907.455,E2 -14907.455} C_VEL
LIN {X 0,Y 326.661,Z 309.789,A -85,B 0,C 180,E1 -14910.341,E2 -14910.341} C_VEL
LIN {X 0,Y 326.691,Z 309.788,A -85,B 0,C 180,E1 -14914.516,E2 -14914.516} C_VEL
LIN {X 0,Y 326.647,Z 309.793,A -85,B 0,C 180,E1 -14918.545,E2 -14918.545} C_VEL
LIN {X 0,Y 326.745,Z 309.778,A -85,B 0,C 180,E1 -14921.177,E2 -14921.177} C_VEL
LIN {X 0,Y 326.763,Z 309.774,A -85,B 0,C 180,E1 -14925.433,E2 -14925.433} C_VEL
LIN {X 0,Y 326.769,Z 309.775,A -85,B 0,C 180,E1 -14928.839,E2 -14928.839} C_VEL
LIN {X 0,Y 326.958,Z 309.751,A -85,B 0,C 180,E1 -14932.59,E2 -14932.59} C_VEL
LIN {X 0,Y 326.775,Z 309.767,A -85,B 0,C 180,E1 -14935.065,E2 -14935.065} C_VEL
LIN {X 0,Y 327.045,Z 309.742,A -85,B 0,C 180,E1 -14937.537,E2 -14937.537} C_VEL
LIN {X 0,Y 327.178,Z 309.721,A -85,B 0,C 180,E1 -14940,E2 -14940} C_VEL
LIN {X 0,Y 327.045,Z 309.736,A -85,B 0,C 180,E1 -14942.463,E2 -14942.463} C_VEL
LIN {X 0,Y 326.968,Z 309.749,A -85,B 0,C 180,E1 -14946.661,E2 -14946.661} C_VEL
LIN {X 0,Y 326.813,Z 309.772,A -85,B 0,C 180,E1 -14949.906,E2 -14949.906} C_VEL
LIN {X 0,Y 326.758,Z 309.778,A -85,B 0,C 180,E1 -14953.685,E2 -14953.685} C_VEL
LIN {X 0,Y 326.699,Z 309.786,A -85,B 0,C 180,E1 -14957.528,E2 -14957.528} C_VEL
LIN {X 0,Y 326.66,Z 309.791,A -85,B 0,C 180,E1 -14960.135,E2 -14960.135} C_VEL
LIN {X 0,Y 326.649,Z 309.792,A -85,B 0,C 180,E1 -14964.129,E2 -14964.129} C_VEL
LIN {X 0,Y 326.682,Z 309.791,A -85,B 0,C 180,E1 -14966.858,E2 -14966.858} C_VEL
LIN {X 0,Y 326.634,Z 309.797,A -85,B 0,C 180,E1 -14970.61,E2 -14970.61} C_VEL
LIN {X 0,Y 326.607,Z 309.796,A -85,B 0,C 180,E1 -14974.019,E2 -14974.019} C_VEL
LIN {X 0,Y 326.627,Z 309.795,A -85,B 0,C 180,E1 -14977.238,E2 -14977.238} C_VEL
LIN {X 0,Y 326.578,Z 309.804,A -85,B 0,C 180,E1 -14981.131,E2 -14981.131} C_VEL
LIN {X 0,Y 326.527,Z 309.809,A -85,B 0,C 180,E1 -14984.743,E2 -14984.743} C_VEL
LIN {X 0,Y 326.576,Z 309.804,A -85,B 0,C 180,E1 -14988.154,E2 -14988.154} C_VEL
LIN {X 0,Y 326.646,Z 309.854,A -85,B 0,C 180,E1 -14991.65,E2 -14991.65} C_VEL
LIN {X 0,Y 328.276,Z 316.336,A -85,B 0,C 180,E1 -14993.764,E2 -14993.764} C_VEL
LIN {X 0,Y 338.118,Z 338.01,A -85,B 0,C 180,E1 -14995.249,E2 -14995.249} C_VEL
LIN {X 0,Y 340.097,Z 343.474,A -85,B 0,C 180,E1 -14995.56,E2 -14995.56} C_VEL
LIN {X 0,Y 340.823,Z 346.704,A -85,B 0,C 180,E1 -14995.701,E2 -14995.701} C_VEL
LIN {X 0,Y 338.702,Z 423.679,A -85,B 0,C 180,E1 -14997.351,E2 -14997.351} C_VEL
LIN {X 0,Y 337.888,Z 437.197,A -85,B 0,C 180,E1 -14997.88,E2 -14997.88} C_VEL
LIN {X 0,Y 337.081,Z 449.027,A -85,B 0,C 180,E1 -14998.584,E2 -14998.584} C_VEL
LIN {X 0,Y 335.894,Z 460.318,A -85,B 0,C 180,E1 -14999.468,E2 -14999.468} C_VEL
LIN {X 0,Y 334.542,Z 471.34,A -85,B 0,C 180,E1 -15000.59,E2 -15000.59} C_VEL
LIN {X 0,Y 332.907,Z 482.222,A -85,B 0,C 180,E1 -15001.984,E2 -15001.984} C_VEL
LIN {X 0,Y 331.329,Z 491.968,A -85,B 0,C 180,E1 -15003.548,E2 -15003.548} C_VEL
LIN {X 0,Y 329.623,Z 501.253,A -85,B 0,C 180,E1 -15005.432,E2 -15005.432} C_VEL
LIN {X 0,Y 328.319,Z 508.685,A -85,B 0,C 180,E1 -15007.337,E2 -15007.337} C_VEL
LIN {X 0,Y 327.207,Z 514.578,A -85,B 0,C 180,E1 -15009.243,E2 -15009.243} C_VEL
LIN {X 0,Y 326.253,Z 519.673,A -85,B 0,C 180,E1 -15011.411,E2 -15011.411} C_VEL
LIN {X 0,Y 325.531,Z 523.516,A -85,B 0,C 180,E1 -15013.7,E2 -15013.7} C_VEL
LIN {X 0,Y 325.27,Z 525.031,A -85,B 0,C 180,E1 -15014.972,E2 -15014.972} C_VEL
LIN {X 0,Y 325.077,Z 526.315,A -85,B 0,C 180,E1 -15016.625,E2 -15016.625} C_VEL
LIN {X 0,Y 324.837,Z 526.98,A -85,B 0,C 180,E1 -15018.771,E2 -15018.771} C_VEL
LIN {X 0,Y 324.775,Z 526.826,A -85,B 0,C 180,E1 -15020.03,E2 -15020.03} C_VEL
LIN {X 0,Y 324.823,Z 526.239,A -85,B 0,C 180,E1 -15021.288,E2 -15021.288} C_VEL
LIN {X 0,Y 324.917,Z 525.264,A -85,B 0,C 180,E1 -15022.543,E2 -15022.543} C_VEL
LIN {X 0,Y 325.1,Z 523.701,A -85,B 0,C 180,E1 -15023.947,E2 -15023.947} C_VEL
LIN {X 0,Y 325.254,Z 519.829,A -85,B 0,C 180,E1 -15026.283,E2 -15026.283} C_VEL
LIN {X 0,Y 325.677,Z 515.563,A -85,B 0,C 180,E1 -15028.144,E2 -15028.144} C_VEL
LIN {X 0,Y 326.268,Z 509.124,A -85,B 0,C 180,E1 -15030.308,E2 -15030.308} C_VEL
LIN {X 0,Y 327.14,Z 502.047,A -85,B 0,C 180,E1 -15032.154,E2 -15032.154} C_VEL
LIN {X 0,Y 328.072,Z 493.257,A -85,B 0,C 180,E1 -15033.992,E2 -15033.992} C_VEL
LIN {X 0,Y 329.138,Z 483.258,A -85,B 0,C 180,E1 -15035.667,E2 -15035.667} C_VEL
LIN {X 0,Y 330.198,Z 473.022,A -85,B 0,C 180,E1 -15037.029,E2 -15037.029} C_VEL
LIN {X 0,Y 331.557,Z 461.604,A -85,B 0,C 180,E1 -15038.225,E2 -15038.225} C_VEL
LIN {X 0,Y 332.401,Z 449.806,A -85,B 0,C 180,E1 -15039.2,E2 -15039.2} C_VEL
LIN {X 0,Y 332.954,Z 436.804,A -85,B 0,C 180,E1 -15039.99,E2 -15039.99} C_VEL
LIN {X 0,Y 333.521,Z 426.043,A -85,B 0,C 180,E1 -15040.432,E2 -15040.432} C_VEL
LIN {X 0,Y 334.067,Z 407.685,A -85,B 0,C 180,E1 -15040.875,E2 -15040.875} C_VEL
LIN {X 0,Y 335.145,Z 343.115,A -85,B 0,C 180,E1 -15042.252,E2 -15042.252} C_VEL
LIN {X 0,Y 332.582,Z 329.453,A -85,B 0,C 180,E1 -15042.713,E2 -15042.713} C_VEL
LIN {X 0,Y 327.968,Z 315.82,A -85,B 0,C 180,E1 -15043.318,E2 -15043.318} C_VEL
LIN {X 0,Y 326.756,Z 309.779,A -85,B 0,C 180,E1 -15045.116,E2 -15045.116} C_VEL
LIN {X 0,Y 326.706,Z 309.788,A -85,B 0,C 180,E1 -15048.824,E2 -15048.824} C_VEL
LIN {X 0,Y 326.595,Z 309.803,A -85,B 0,C 180,E1 -15052.788,E2 -15052.788} C_VEL
LIN {X 0,Y 326.63,Z 309.795,A -85,B 0,C 180,E1 -15055.488,E2 -15055.488} C_VEL
LIN {X 0,Y 326.612,Z 309.797,A -85,B 0,C 180,E1 -15059.663,E2 -15059.663} C_VEL
LIN {X 0,Y 326.599,Z 309.799,A -85,B 0,C 180,E1 -15060.05,E2 -15060.05} C_VEL
LIN {X 0,Y 325.922,Z 309.889,A -85,B 0,C 180,E1 -15061.079,E2 -15061.079} C_VEL
LIN {X 0,Y 323.046,Z 310.249,A -85,B 0,C 180,E1 -15062.754,E2 -15062.754} C_VEL
LIN {X 0,Y 320.636,Z 310.547,A -85,B 0,C 180,E1 -15064.112,E2 -15064.112} C_VEL
LIN {X 0,Y 319.637,Z 310.669,A -85,B 0,C 180,E1 -15065.163,E2 -15065.163} C_VEL
LIN {X 0,Y 319.574,Z 310.675,A -85,B 0,C 180,E1 -15065.519,E2 -15065.519} C_VEL
LIN {X 0,Y 319.54,Z 310.679,A -85,B 0,C 180,E1 -15069.629,E2 -15069.629} C_VEL
LIN {X 0,Y 319.515,Z 310.681,A -85,B 0,C 180,E1 -15073.459,E2 -15073.459} C_VEL
LIN {X 0,Y 319.548,Z 310.681,A -85,B 0,C 180,E1 -15077.016,E2 -15077.016} C_VEL
LIN {X 0,Y 319.539,Z 310.676,A -85,B 0,C 180,E1 -15080.37,E2 -15080.37} C_VEL
LIN {X 0,Y 319.573,Z 310.674,A -85,B 0,C 180,E1 -15084.457,E2 -15084.457} C_VEL
LIN {X 0,Y 319.525,Z 310.679,A -85,B 0,C 180,E1 -15088.138,E2 -15088.138} C_VEL
LIN {X 0,Y 319.609,Z 310.673,A -85,B 0,C 180,E1 -15091.588,E2 -15091.588} C_VEL
LIN {X 0,Y 319.596,Z 310.674,A -85,B 0,C 180,E1 -15095.303,E2 -15095.303} C_VEL
LIN {X 0,Y 319.596,Z 310.671,A -85,B 0,C 180,E1 -15099.4,E2 -15099.4} C_VEL
LIN {X 0,Y 319.651,Z 310.667,A -85,B 0,C 180,E1 -15102.073,E2 -15102.073} C_VEL
LIN {X 0,Y 319.725,Z 310.66,A -85,B 0,C 180,E1 -15106.008,E2 -15106.008} C_VEL
LIN {X 0,Y 319.744,Z 310.654,A -85,B 0,C 180,E1 -15109.873,E2 -15109.873} C_VEL
LIN {X 0,Y 319.903,Z 310.634,A -85,B 0,C 180,E1 -15113.694,E2 -15113.694} C_VEL
LIN {X 0,Y 319.982,Z 310.623,A -85,B 0,C 180,E1 -15117.482,E2 -15117.482} C_VEL
LIN {X 0,Y 320.123,Z 310.606,A -85,B 0,C 180,E1 -15120,E2 -15120} C_VEL
LIN {X 0,Y 319.982,Z 310.627,A -85,B 0,C 180,E1 -15122.518,E2 -15122.518} C_VEL
LIN {X 0,Y 319.938,Z 310.633,A -85,B 0,C 180,E1 -15126.306,E2 -15126.306} C_VEL
LIN {X 0,Y 319.835,Z 310.642,A -85,B 0,C 180,E1 -15128.848,E2 -15128.848} C_VEL
LIN {X 0,Y 319.675,Z 310.665,A -85,B 0,C 180,E1 -15132.7,E2 -15132.7} C_VEL
LIN {X 0,Y 319.692,Z 310.66,A -85,B 0,C 180,E1 -15135.296,E2 -15135.296} C_VEL
LIN {X 0,Y 319.667,Z 310.665,A -85,B 0,C 180,E1 -15139.256,E2 -15139.256} C_VEL
LIN {X 0,Y 319.564,Z 310.678,A -85,B 0,C 180,E1 -15143.32,E2 -15143.32} C_VEL
LIN {X 0,Y 319.629,Z 310.667,A -85,B 0,C 180,E1 -15146.089,E2 -15146.089} C_VEL
LIN {X 0,Y 319.585,Z 310.678,A -85,B 0,C 180,E1 -15148.934,E2 -15148.934} C_VEL
LIN {X 0,Y 319.534,Z 310.68,A -85,B 0,C 180,E1 -15151.862,E2 -15151.862} C_VEL
LIN {X 0,Y 319.576,Z 310.678,A -85,B 0,C 180,E1 -15155.544,E2 -15155.544} C_VEL
LIN {X 0,Y 319.569,Z 310.676,A -85,B 0,C 180,E1 -15158.009,E2 -15158.009} C_VEL
LIN {X 0,Y 319.522,Z 310.686,A -85,B 0,C 180,E1 -15161.598,E2 -15161.598} C_VEL
LIN {X 0,Y 319.485,Z 310.689,A -85,B 0,C 180,E1 -15165.258,E2 -15165.258} C_VEL
LIN {X 0,Y 319.525,Z 310.681,A -85,B 0,C 180,E1 -15168.713,E2 -15168.713} C_VEL
LIN {X 0,Y 319.559,Z 310.677,A -85,B 0,C 180,E1 -15172.349,E2 -15172.349} C_VEL
LIN {X 0,Y 319.558,Z 310.678,A -85,B 0,C 180,E1 -15175.124,E2 -15175.124} C_VEL
LIN {X 0,Y 319.599,Z 310.863,A -85,B 0,C 180,E1 -15179.05,E2 -15179.05} C_VEL
LIN {X 0,Y 321.865,Z 321.329,A -85,B 0,C 180,E1 -15182.002,E2 -15182.002} C_VEL
LIN {X 0,Y 323.308,Z 329.558,A -85,B 0,C 180,E1 -15184.231,E2 -15184.231} C_VEL
LIN {X 0,Y 322.492,Z 338.011,A -85,B 0,C 180,E1 -15186.343,E2 -15186.343} C_VEL
LIN {X 0,Y 328.005,Z 378.104,A -85,B 0,C 180,E1 -15187.616,E2 -15187.616} C_VEL
LIN {X 0,Y 326.691,Z 446.612,A -85,B 0,C 180,E1 -15189.128,E2 -15189.128} C_VEL
LIN {X 0,Y 325.925,Z 459.908,A -85,B 0,C 180,E1 -15189.654,E2 -15189.654} C_VEL
LIN {X 0,Y 324.995,Z 472.692,A -85,B 0,C 180,E1 -15190.417,E2 -15190.417} C_VEL
LIN {X 0,Y 324.008,Z 484.039,A -85,B 0,C 180,E1 -15191.342,E2 -15191.342} C_VEL
LIN {X 0,Y 322.882,Z 494.447,A -85,B 0,C 180,E1 -15192.423,E2 -15192.423} C_VEL
LIN {X 0,Y 321.773,Z 505.122,A -85,B 0,C 180,E1 -15193.817,E2 -15193.817} C_VEL
LIN {X 0,Y 320.685,Z 514.911,A -85,B 0,C 180,E1 -15195.403,E2 -15195.403} C_VEL
LIN {X 0,Y 319.766,Z 522.836,A -85,B 0,C 180,E1 -15196.982,E2 -15196.982} C_VEL
LIN {X 0,Y 318.863,Z 530.555,A -85,B 0,C 180,E1 -15198.881,E2 -15198.881} C_VEL
LIN {X 0,Y 318.289,Z 537.678,A -85,B 0,C 180,E1 -15201.109,E2 -15201.109} C_VEL
LIN {X 0,Y 317.978,Z 542.395,A -85,B 0,C 180,E1 -15203.019,E2 -15203.019} C_VEL
LIN {X 0,Y 317.83,Z 545.979,A -85,B 0,C 180,E1 -15204.926,E2 -15204.926} C_VEL
LIN {X 0,Y 317.844,Z 547.81,A -85,B 0,C 180,E1 -15206.197,E2 -15206.197} C_VEL
LIN {X 0,Y 317.8,Z 549.175,A -85,B 0,C 180,E1 -15207.466,E2 -15207.466} C_VEL
LIN {X 0,Y 317.81,Z 550.143,A -85,B 0,C 180,E1 -15208.734,E2 -15208.734} C_VEL
LIN {X 0,Y 317.853,Z 550.718,A -85,B 0,C 180,E1 -15210.001,E2 -15210.001} C_VEL
LIN {X 0,Y 317.781,Z 550.878,A -85,B 0,C 180,E1 -15211.268,E2 -15211.268} C_VEL
LIN {X 0,Y 317.778,Z 550.617,A -85,B 0,C 180,E1 -15212.536,E2 -15212.536} C_VEL
LIN {X 0,Y 317.809,Z 549.971,A -85,B 0,C 180,E1 -15213.805,E2 -15213.805} C_VEL
LIN {X 0,Y 317.842,Z 548.245,A -85,B 0,C 180,E1 -15215.715,E2 -15215.715} C_VEL
LIN {X 0,Y 318.214,Z 544.516,A -85,B 0,C 180,E1 -15218.254,E2 -15218.254} C_VEL
LIN {X 0,Y 318.773,Z 540.509,A -85,B 0,C 180,E1 -15220.159,E2 -15220.159} C_VEL
LIN {X 0,Y 319.734,Z 534.376,A -85,B 0,C 180,E1 -15222.376,E2 -15222.376} C_VEL
LIN {X 0,Y 321.042,Z 527.708,A -85,B 0,C 180,E1 -15224.258,E2 -15224.258} C_VEL
LIN {X 0,Y 322.455,Z 519.46,A -85,B 0,C 180,E1 -15226.135,E2 -15226.135} C_VEL
LIN {X 0,Y 323.966,Z 511.032,A -85,B 0,C 180,E1 -15227.681,E2 -15227.681} C_VEL
LIN {X 0,Y 325.75,Z 500.647,A -85,B 0,C 180,E1 -15229.209,E2 -15229.209} C_VEL
LIN {X 0,Y 327.41,Z 490.399,A -85,B 0,C 180,E1 -15230.415,E2 -15230.415} C_VEL
LIN {X 0,Y 329.008,Z 479.202,A -85,B 0,C 180,E1 -15231.458,E2 -15231.458} C_VEL
LIN {X 0,Y 330.395,Z 466.626,A -85,B 0,C 180,E1 -15232.348,E2 -15232.348} C_VEL
LIN {X 0,Y 331.605,Z 453.169,A -85,B 0,C 180,E1 -15233.002,E2 -15233.002} C_VEL
LIN {X 0,Y 332.253,Z 439.796,A -85,B 0,C 180,E1 -15233.408,E2 -15233.408} C_VEL
LIN {X 0,Y 333.678,Z 379.346,A -85,B 0,C 180,E1 -15234.727,E2 -15234.727} C_VEL
LIN {X 0,Y 330.572,Z 361.015,A -85,B 0,C 180,E1 -15235.46,E2 -15235.46} C_VEL
LIN {X 0,Y 325.721,Z 338.422,A -85,B 0,C 180,E1 -15236.493,E2 -15236.493} C_VEL
LIN {X 0,Y 325.527,Z 337.384,A -85,B 0,C 180,E1 -15236.548,E2 -15236.548} C_VEL
LIN {X 0,Y 323.903,Z 328.556,A -85,B 0,C 180,E1 -15239.112,E2 -15239.112} C_VEL
LIN {X 0,Y 321.385,Z 317.932,A -85,B 0,C 180,E1 -15242.395,E2 -15242.395} C_VEL
LIN {X 0,Y 319.619,Z 310.674,A -85,B 0,C 180,E1 -15244.776,E2 -15244.776} C_VEL
LIN {X 0,Y 319.545,Z 310.681,A -85,B 0,C 180,E1 -15248.012,E2 -15248.012} C_VEL
LIN {X 0,Y 319.527,Z 310.684,A -85,B 0,C 180,E1 -15251.597,E2 -15251.597} C_VEL
LIN {X 0,Y 319.489,Z 310.688,A -85,B 0,C 180,E1 -15255.257,E2 -15255.257} C_VEL
LIN {X 0,Y 319.53,Z 310.684,A -85,B 0,C 180,E1 -15258.712,E2 -15258.712} C_VEL
LIN {X 0,Y 319.555,Z 310.677,A -85,B 0,C 180,E1 -15262.349,E2 -15262.349} C_VEL
LIN {X 0,Y 319.561,Z 310.675,A -85,B 0,C 180,E1 -15265.123,E2 -15265.123} C_VEL
LIN {X 0,Y 319.571,Z 310.673,A -85,B 0,C 180,E1 -15269.058,E2 -15269.058} C_VEL
LIN {X 0,Y 319.609,Z 310.671,A -85,B 0,C 180,E1 -15272.498,E2 -15272.498} C_VEL
LIN {X 0,Y 319.606,Z 310.675,A -85,B 0,C 180,E1 -15275.304,E2 -15275.304} C_VEL
LIN {X 0,Y 319.597,Z 310.671,A -85,B 0,C 180,E1 -15278.048,E2 -15278.048} C_VEL
LIN {X 0,Y 319.69,Z 310.657,A -85,B 0,C 180,E1 -15280.962,E2 -15280.962} C_VEL
LIN {X 0,Y 319.731,Z 310.65,A -85,B 0,C 180,E1 -15285.276,E2 -15285.276} C_VEL
LIN {X 0,Y 319.752,Z 310.644,A -85,B 0,C 180,E1 -15289.872,E2 -15289.872} C_VEL
LIN {X 0,Y 319.912,Z 310.629,A -85,B 0,C 180,E1 -15292.426,E2 -15292.426} C_VEL
LIN {X 0,Y 319.745,Z 310.643,A -85,B 0,C 180,E1 -15294.956,E2 -15294.956} C_VEL
LIN {X 0,Y 319.989,Z 310.621,A -85,B 0,C 180,E1 -15297.482,E2 -15297.482} C_VEL
LIN {X 0,Y 320.13,Z 310.598,A -85,B 0,C 180,E1 -15300,E2 -15300} C_VEL
LIN {X 0,Y 319.989,Z 310.615,A -85,B 0,C 180,E1 -15302.517,E2 -15302.517} C_VEL
LIN {X 0,Y 319.929,Z 310.625,A -85,B 0,C 180,E1 -15306.652,E2 -15306.652} C_VEL
LIN {X 0,Y 319.757,Z 310.653,A -85,B 0,C 180,E1 -15310.127,E2 -15310.127} C_VEL
LIN {X 0,Y 319.731,Z 310.657,A -85,B 0,C 180,E1 -15314.724,E2 -15314.724} C_VEL
LIN {X 0,Y 319.689,Z 310.662,A -85,B 0,C 180,E1 -15319.038,E2 -15319.038} C_VEL
LIN {X 0,Y 319.56,Z 310.676,A -85,B 0,C 180,E1 -15323.32,E2 -15323.32} C_VEL
LIN {X 0,Y 319.634,Z 310.666,A -85,B 0,C 180,E1 -15326.088,E2 -15326.088} C_VEL
LIN {X 0,Y 319.58,Z 310.67,A -85,B 0,C 180,E1 -15328.934,E2 -15328.934} C_VEL
LIN {X 0,Y 319.53,Z 310.675,A -85,B 0,C 180,E1 -15331.862,E2 -15331.862} C_VEL
LIN {X 0,Y 319.58,Z 310.674,A -85,B 0,C 180,E1 -15335.543,E2 -15335.543} C_VEL
LIN {X 0,Y 319.557,Z 310.676,A -85,B 0,C 180,E1 -15338.01,E2 -15338.01} C_VEL
LIN {X 0,Y 319.526,Z 310.685,A -85,B 0,C 180,E1 -15341.597,E2 -15341.597} C_VEL
LIN {X 0,Y 319.488,Z 310.687,A -85,B 0,C 180,E1 -15345.257,E2 -15345.257} C_VEL
LIN {X 0,Y 319.528,Z 310.682,A -85,B 0,C 180,E1 -15348.712,E2 -15348.712} C_VEL
LIN {X 0,Y 319.581,Z 310.751,A -85,B 0,C 180,E1 -15351.037,E2 -15351.037} C_VEL
LIN {X 0,Y 321.179,Z 316.93,A -85,B 0,C 180,E1 -15353.046,E2 -15353.046} C_VEL
LIN {X 0,Y 329.23,Z 333.926,A -85,B 0,C 180,E1 -15354.301,E2 -15354.301} C_VEL
LIN {X 0,Y 334.046,Z 345.599,A -85,B 0,C 180,E1 -15355.051,E2 -15355.051} C_VEL
LIN {X 0,Y 334.579,Z 348.786,A -85,B 0,C 180,E1 -15355.177,E2 -15355.177} C_VEL
LIN {X 0,Y 332.34,Z 424.404,A -85,B 0,C 180,E1 -15356.826,E2 -15356.826} C_VEL
LIN {X 0,Y 331.488,Z 437.763,A -85,B 0,C 180,E1 -15357.363,E2 -15357.363} C_VEL
LIN {X 0,Y 330.541,Z 450.636,A -85,B 0,C 180,E1 -15358.158,E2 -15358.158} C_VEL
LIN {X 0,Y 329.16,Z 462.773,A -85,B 0,C 180,E1 -15359.174,E2 -15359.174} C_VEL
LIN {X 0,Y 327.615,Z 474.369,A -85,B 0,C 180,E1 -15360.436,E2 -15360.436} C_VEL
LIN {X 0,Y 325.902,Z 484.963,A -85,B 0,C 180,E1 -15361.898,E2 -15361.898} C_VEL
LIN {X 0,Y 324.147,Z 494.803,A -85,B 0,C 180,E1 -15363.61,E2 -15363.61} C_VEL
LIN {X 0,Y 322.702,Z 502.262,A -85,B 0,C 180,E1 -15365.213,E2 -15365.213} C_VEL
LIN {X 0,Y 321.356,Z 509.549,A -85,B 0,C 180,E1 -15367.158,E2 -15367.158} C_VEL
LIN {X 0,Y 320.369,Z 514.428,A -85,B 0,C 180,E1 -15368.779,E2 -15368.779} C_VEL
LIN {X 0,Y 319.446,Z 519.121,A -85,B 0,C 180,E1 -15370.73,E2 -15370.73} C_VEL
LIN {X 0,Y 318.949,Z 521.582,A -85,B 0,C 180,E1 -15372.031,E2 -15372.031} C_VEL
LIN {X 0,Y 318.537,Z 523.575,A -85,B 0,C 180,E1 -15373.332,E2 -15373.332} C_VEL
LIN {X 0,Y 318.242,Z 525.14,A -85,B 0,C 180,E1 -15374.632,E2 -15374.632} C_VEL
LIN {X 0,Y 318.009,Z 526.602,A -85,B 0,C 180,E1 -15376.507,E2 -15376.507} C_VEL
LIN {X 0,Y 317.774,Z 527.228,A -85,B 0,C 180,E1 -15378.518,E2 -15378.518} C_VEL
LIN {X 0,Y 317.681,Z 527.133,A -85,B 0,C 180,E1 -15379.805,E2 -15379.805} C_VEL
LIN {X 0,Y 317.728,Z 526.598,A -85,B 0,C 180,E1 -15381.092,E2 -15381.092} C_VEL
LIN {X 0,Y 317.815,Z 525.66,A -85,B 0,C 180,E1 -15382.375,E2 -15382.375} C_VEL
LIN {X 0,Y 318.028,Z 523.967,A -85,B 0,C 180,E1 -15383.956,E2 -15383.956} C_VEL
LIN {X 0,Y 318.169,Z 520.378,A -85,B 0,C 180,E1 -15386.2,E2 -15386.2} C_VEL
LIN {X 0,Y 318.584,Z 516.196,A -85,B 0,C 180,E1 -15388.103,E2 -15388.103} C_VEL
LIN {X 0,Y 319.164,Z 509.852,A -85,B 0,C 180,E1 -15390.315,E2 -15390.315} C_VEL
LIN {X 0,Y 320.065,Z 502.923,A -85,B 0,C 180,E1 -15392.202,E2 -15392.202} C_VEL
LIN {X 0,Y 321.017,Z 494.264,A -85,B 0,C 180,E1 -15394.079,E2 -15394.079} C_VEL
LIN {X 0,Y 322.026,Z 485.401,A -85,B 0,C 180,E1 -15395.635,E2 -15395.635} C_VEL
LIN {X 0,Y 323.1,Z 475.66,A -85,B 0,C 180,E1 -15397.027,E2 -15397.027} C_VEL
LIN {X 0,Y 324.261,Z 466.352,A -85,B 0,C 180,E1 -15398.098,E2 -15398.098} C_VEL
LIN {X 0,Y 325.257,Z 454.849,A -85,B 0,C 180,E1 -15399.169,E2 -15399.169} C_VEL
LIN {X 0,Y 325.99,Z 442.956,A -85,B 0,C 180,E1 -15400.009,E2 -15400.009} C_VEL
LIN {X 0,Y 326.47,Z 430.145,A -85,B 0,C 180,E1 -15400.66,E2 -15400.66} C_VEL
LIN {X 0,Y 327.037,Z 419.405,A -85,B 0,C 180,E1 -15400.994,E2 -15400.994} C_VEL
LIN {X 0,Y 328.557,Z 344.85,A -85,B 0,C 180,E1 -15402.61,E2 -15402.61} C_VEL
LIN {X 0,Y 326.09,Z 331.544,A -85,B 0,C 180,E1 -15403.068,E2 -15403.068} C_VEL
LIN {X 0,Y 320.788,Z 316.07,A -85,B 0,C 180,E1 -15403.785,E2 -15403.785} C_VEL
LIN {X 0,Y 319.688,Z 310.659,A -85,B 0,C 180,E1 -15405.458,E2 -15405.458} C_VEL
LIN {X 0,Y 319.627,Z 310.668,A -85,B 0,C 180,E1 -15409.257,E2 -15409.257} C_VEL
LIN {X 0,Y 319.549,Z 310.677,A -85,B 0,C 180,E1 -15413.32,E2 -15413.32} C_VEL
LIN {X 0,Y 319.564,Z 310.676,A -85,B 0,C 180,E1 -15416.093,E2 -15416.093} C_VEL
LIN {X 0,Y 319.538,Z 310.682,A -85,B 0,C 180,E1 -15418.937,E2 -15418.937} C_VEL
LIN {X 0,Y 319.52,Z 310.68,A -85,B 0,C 180,E1 -15421.862,E2 -15421.862} C_VEL
LIN {X 0,Y 319.574,Z 310.675,A -85,B 0,C 180,E1 -15425.519,E2 -15425.519} C_VEL
LIN {X 0,Y 318.945,Z 310.756,A -85,B 0,C 180,E1 -15426.571,E2 -15426.571} C_VEL
LIN {X 0,Y 316.061,Z 311.115,A -85,B 0,C 180,E1 -15428.282,E2 -15428.282} C_VEL
LIN {X 0,Y 313.583,Z 311.424,A -85,B 0,C 180,E1 -15429.669,E2 -15429.669} C_VEL
LIN {X 0,Y 312.511,Z 311.557,A -85,B 0,C 180,E1 -15430.744,E2 -15430.744} C_VEL
LIN {X 0,Y 312.422,Z 311.565,A -85,B 0,C 180,E1 -15431.109,E2 -15431.109} C_VEL
LIN {X 0,Y 312.446,Z 311.559,A -85,B 0,C 180,E1 -15434.209,E2 -15434.209} C_VEL
LIN {X 0,Y 312.477,Z 311.558,A -85,B 0,C 180,E1 -15437.918,E2 -15437.918} C_VEL
LIN {X 0,Y 312.489,Z 311.557,A -85,B 0,C 180,E1 -15440.97,E2 -15440.97} C_VEL
LIN {X 0,Y 312.524,Z 311.552,A -85,B 0,C 180,E1 -15444.219,E2 -15444.219} C_VEL
LIN {X 0,Y 312.498,Z 311.56,A -85,B 0,C 180,E1 -15447.333,E2 -15447.333} C_VEL
LIN {X 0,Y 312.545,Z 311.549,A -85,B 0,C 180,E1 -15451.276,E2 -15451.276} C_VEL
LIN {X 0,Y 312.578,Z 311.546,A -85,B 0,C 180,E1 -15454.71,E2 -15454.71} C_VEL
LIN {X 0,Y 312.531,Z 311.548,A -85,B 0,C 180,E1 -15458.912,E2 -15458.912} C_VEL
LIN {X 0,Y 312.631,Z 311.54,A -85,B 0,C 180,E1 -15461.656,E2 -15461.656} C_VEL
LIN {X 0,Y 312.686,Z 311.536,A -85,B 0,C 180,E1 -15465.686,E2 -15465.686} C_VEL
LIN {X 0,Y 312.69,Z 311.53,A -85,B 0,C 180,E1 -15469.642,E2 -15469.642} C_VEL
LIN {X 0,Y 312.81,Z 311.52,A -85,B 0,C 180,E1 -15472.253,E2 -15472.253} C_VEL
LIN {X 0,Y 312.7,Z 311.531,A -85,B 0,C 180,E1 -15474.842,E2 -15474.842} C_VEL
LIN {X 0,Y 312.981,Z 311.494,A -85,B 0,C 180,E1 -15478.713,E2 -15478.713} C_VEL
LIN {X 0,Y 312.982,Z 311.491,A -85,B 0,C 180,E1 -15481.287,E2 -15481.287} C_VEL
LIN {X 0,Y 312.708,Z 311.53,A -85,B 0,C 180,E1 -15485.158,E2 -15485.158} C_VEL
LIN {X 0,Y 312.859,Z 311.51,A -85,B 0,C 180,E1 -15487.746,E2 -15487.746} C_VEL
LIN {X 0,Y 312.662,Z 311.531,A -85,B 0,C 180,E1 -15491.672,E2 -15491.672} C_VEL
LIN {X 0,Y 312.693,Z 311.536,A -85,B 0,C 180,E1 -15494.888,E2 -15494.888} C_VEL
LIN {X 0,Y 312.623,Z 311.542,A -85,B 0,C 180,E1 -15499.237,E2 -15499.237} C_VEL
LIN {X 0,Y 312.54,Z 311.554,A -85,B 0,C 180,E1 -15502.79,E2 -15502.79} C_VEL
LIN {X 0,Y 312.597,Z 311.543,A -85,B 0,C 180,E1 -15505.936,E2 -15505.936} C_VEL
LIN {X 0,Y 312.541,Z 311.551,A -85,B 0,C 180,E1 -15509.651,E2 -15509.651} C_VEL
LIN {X 0,Y 312.515,Z 311.556,A -85,B 0,C 180,E1 -15513.69,E2 -15513.69} C_VEL
LIN {X 0,Y 312.533,Z 311.558,A -85,B 0,C 180,E1 -15517.384,E2 -15517.384} C_VEL
LIN {X 0,Y 312.486,Z 311.558,A -85,B 0,C 180,E1 -15520.71,E2 -15520.71} C_VEL
LIN {X 0,Y 312.448,Z 311.563,A -85,B 0,C 180,E1 -15524.211,E2 -15524.211} C_VEL
LIN {X 0,Y 312.481,Z 311.561,A -85,B 0,C 180,E1 -15527.92,E2 -15527.92} C_VEL
LIN {X 0,Y 312.532,Z 311.556,A -85,B 0,C 180,E1 -15531.912,E2 -15531.912} C_VEL
LIN {X 0,Y 312.504,Z 311.561,A -85,B 0,C 180,E1 -15535.791,E2 -15535.791} C_VEL
LIN {X 0,Y 312.543,Z 311.745,A -85,B 0,C 180,E1 -15538.704,E2 -15538.704} C_VEL
LIN {X 0,Y 314.784,Z 322.065,A -85,B 0,C 180,E1 -15541.688,E2 -15541.688} C_VEL
LIN {X 0,Y 316.256,Z 330.272,A -85,B 0,C 180,E1 -15543.968,E2 -15543.968} C_VEL
LIN {X 0,Y 316.228,Z 332.961,A -85,B 0,C 180,E1 -15544.672,E2 -15544.672} C_VEL
LIN {X 0,Y 315.657,Z 337.91,A -85,B 0,C 180,E1 -15545.903,E2 -15545.903} C_VEL
LIN {X 0,Y 321.286,Z 378.539,A -85,B 0,C 180,E1 -15547.222,E2 -15547.222} C_VEL
LIN {X 0,Y 319.941,Z 446.433,A -85,B 0,C 180,E1 -15548.75,E2 -15548.75} C_VEL
LIN {X 0,Y 319.152,Z 459.701,A -85,B 0,C 180,E1 -15549.287,E2 -15549.287} C_VEL
LIN {X 0,Y 318.2,Z 472.471,A -85,B 0,C 180,E1 -15550.065,E2 -15550.065} C_VEL
LIN {X 0,Y 317.072,Z 484.6,A -85,B 0,C 180,E1 -15551.086,E2 -15551.086} C_VEL
LIN {X 0,Y 315.724,Z 496.156,A -85,B 0,C 180,E1 -15552.346,E2 -15552.346} C_VEL
LIN {X 0,Y 314.663,Z 506.355,A -85,B 0,C 180,E1 -15553.752,E2 -15553.752} C_VEL
LIN {X 0,Y 313.543,Z 515.935,A -85,B 0,C 180,E1 -15555.395,E2 -15555.395} C_VEL
LIN {X 0,Y 312.468,Z 524.995,A -85,B 0,C 180,E1 -15557.333,E2 -15557.333} C_VEL
LIN {X 0,Y 311.668,Z 532.281,A -85,B 0,C 180,E1 -15559.279,E2 -15559.279} C_VEL
LIN {X 0,Y 311.226,Z 537.193,A -85,B 0,C 180,E1 -15560.906,E2 -15560.906} C_VEL
LIN {X 0,Y 310.906,Z 541.957,A -85,B 0,C 180,E1 -15562.859,E2 -15562.859} C_VEL
LIN {X 0,Y 310.744,Z 545.586,A -85,B 0,C 180,E1 -15564.81,E2 -15564.81} C_VEL
LIN {X 0,Y 310.753,Z 547.453,A -85,B 0,C 180,E1 -15566.11,E2 -15566.11} C_VEL
LIN {X 0,Y 310.721,Z 548.843,A -85,B 0,C 180,E1 -15567.408,E2 -15567.408} C_VEL
LIN {X 0,Y 310.721,Z 549.83,A -85,B 0,C 180,E1 -15568.705,E2 -15568.705} C_VEL
LIN {X 0,Y 310.759,Z 550.425,A -85,B 0,C 180,E1 -15570.001,E2 -15570.001} C_VEL
LIN {X 0,Y 310.693,Z 550.618,A -85,B 0,C 180,E1 -15571.297,E2 -15571.297} C_VEL
LIN {X 0,Y 310.7,Z 550.381,A -85,B 0,C 180,E1 -15572.594,E2 -15572.594} C_VEL
LIN {X 0,Y 310.72,Z 549.753,A -85,B 0,C 180,E1 -15573.891,E2 -15573.891} C_VEL
LIN {X 0,Y 310.83,Z 547.328,A -85,B 0,C 180,E1 -15576.492,E2 -15576.492} C_VEL
LIN {X 0,Y 311.157,Z 544.381,A -85,B 0,C 180,E1 -15578.443,E2 -15578.443} C_VEL
LIN {X 0,Y 311.746,Z 540.414,A -85,B 0,C 180,E1 -15580.391,E2 -15580.391} C_VEL
LIN {X 0,Y 312.602,Z 535.333,A -85,B 0,C 180,E1 -15582.333,E2 -15582.333} C_VEL
LIN {X 0,Y 313.904,Z 528.972,A -85,B 0,C 180,E1 -15584.258,E2 -15584.258} C_VEL
LIN {X 0,Y 315.376,Z 521.065,A -85,B 0,C 180,E1 -15586.17,E2 -15586.17} C_VEL
LIN {X 0,Y 316.857,Z 512.995,A -85,B 0,C 180,E1 -15587.757,E2 -15587.757} C_VEL
LIN {X 0,Y 318.66,Z 503.196,A -85,B 0,C 180,E1 -15589.319,E2 -15589.319} C_VEL
LIN {X 0,Y 320.581,Z 492.264,A -85,B 0,C 180,E1 -15590.702,E2 -15590.702} C_VEL
LIN {X 0,Y 322.195,Z 481.578,A -85,B 0,C 180,E1 -15591.766,E2 -15591.766} C_VEL
LIN {X 0,Y 323.773,Z 468.734,A -85,B 0,C 180,E1 -15592.746,E2 -15592.746} C_VEL
LIN {X 0,Y 324.989,Z 456.511,A -85,B 0,C 180,E1 -15593.414,E2 -15593.414} C_VEL
LIN {X 0,Y 325.811,Z 444.052,A -85,B 0,C 180,E1 -15593.857,E2 -15593.857} C_VEL
LIN {X 0,Y 327.422,Z 380.449,A -85,B 0,C 180,E1 -15595.284,E2 -15595.284} C_VEL
LIN {X 0,Y 324.354,Z 362.358,A -85,B 0,C 180,E1 -15596.032,E2 -15596.032} C_VEL
LIN {X 0,Y 319.965,Z 341.44,A -85,B 0,C 180,E1 -15597.01,E2 -15597.01} C_VEL
LIN {X 0,Y 318.392,Z 336.986,A -85,B 0,C 180,E1 -15597.321,E2 -15597.321} C_VEL
LIN {X 0,Y 316.398,Z 327.304,A -85,B 0,C 180,E1 -15600.256,E2 -15600.256} C_VEL
LIN {X 0,Y 314.134,Z 318.023,A -85,B 0,C 180,E1 -15603.239,E2 -15603.239} C_VEL
LIN {X 0,Y 312.554,Z 311.553,A -85,B 0,C 180,E1 -15605.48,E2 -15605.48} C_VEL
LIN {X 0,Y 312.5,Z 311.56,A -85,B 0,C 180,E1 -15609.029,E2 -15609.029} C_VEL
LIN {X 0,Y 312.491,Z 311.558,A -85,B 0,C 180,E1 -15612.432,E2 -15612.432} C_VEL
LIN {X 0,Y 312.459,Z 311.565,A -85,B 0,C 180,E1 -15616.035,E2 -15616.035} C_VEL
LIN {X 0,Y 312.505,Z 311.552,A -85,B 0,C 180,E1 -15619.874,E2 -15619.874} C_VEL
LIN {X 0,Y 312.536,Z 311.551,A -85,B 0,C 180,E1 -15624.05,E2 -15624.05} C_VEL
LIN {X 0,Y 312.505,Z 311.558,A -85,B 0,C 180,E1 -15627.334,E2 -15627.334} C_VEL
LIN {X 0,Y 312.553,Z 311.554,A -85,B 0,C 180,E1 -15631.276,E2 -15631.276} C_VEL
LIN {X 0,Y 312.586,Z 311.546,A -85,B 0,C 180,E1 -15634.711,E2 -15634.711} C_VEL
LIN {X 0,Y 312.588,Z 311.542,A -85,B 0,C 180,E1 -15637.529,E2 -15637.529} C_VEL
LIN {X 0,Y 312.639,Z 311.534,A -85,B 0,C 180,E1 -15641.656,E2 -15641.656} C_VEL
LIN {X 0,Y 312.694,Z 311.525,A -85,B 0,C 180,E1 -15645.686,E2 -15645.686} C_VEL
LIN {X 0,Y 312.698,Z 311.523,A -85,B 0,C 180,E1 -15649.642,E2 -15649.642} C_VEL
LIN {X 0,Y 312.853,Z 311.509,A -85,B 0,C 180,E1 -15652.254,E2 -15652.254} C_VEL
LIN {X 0,Y 312.715,Z 311.518,A -85,B 0,C 180,E1 -15654.842,E2 -15654.842} C_VEL
LIN {X 0,Y 312.988,Z 311.482,A -85,B 0,C 180,E1 -15658.713,E2 -15658.713} C_VEL
LIN {X 0,Y 312.988,Z 311.491,A -85,B 0,C 180,E1 -15661.286,E2 -15661.286} C_VEL
LIN {X 0,Y 312.716,Z 311.525,A -85,B 0,C 180,E1 -15665.157,E2 -15665.157} C_VEL
LIN {X 0,Y 312.872,Z 311.502,A -85,B 0,C 180,E1 -15667.746,E2 -15667.746} C_VEL
LIN {X 0,Y 312.668,Z 311.531,A -85,B 0,C 180,E1 -15671.671,E2 -15671.671} C_VEL
LIN {X 0,Y 312.7,Z 311.532,A -85,B 0,C 180,E1 -15674.887,E2 -15674.887} C_VEL
LIN {X 0,Y 312.629,Z 311.54,A -85,B 0,C 180,E1 -15679.236,E2 -15679.236} C_VEL
LIN {X 0,Y 312.526,Z 311.556,A -85,B 0,C 180,E1 -15682.78,E2 -15682.78} C_VEL
LIN {X 0,Y 312.602,Z 311.542,A -85,B 0,C 180,E1 -15685.935,E2 -15685.935} C_VEL
LIN {X 0,Y 312.538,Z 311.551,A -85,B 0,C 180,E1 -15689.651,E2 -15689.651} C_VEL
LIN {X 0,Y 312.519,Z 311.552,A -85,B 0,C 180,E1 -15693.689,E2 -15693.689} C_VEL
LIN {X 0,Y 312.525,Z 311.551,A -85,B 0,C 180,E1 -15697.385,E2 -15697.385} C_VEL
LIN {X 0,Y 312.49,Z 311.555,A -85,B 0,C 180,E1 -15700.709,E2 -15700.709} C_VEL
LIN {X 0,Y 312.452,Z 311.564,A -85,B 0,C 180,E1 -15704.21,E2 -15704.21} C_VEL
LIN {X 0,Y 312.484,Z 311.561,A -85,B 0,C 180,E1 -15707.919,E2 -15707.919} C_VEL
LIN {X 0,Y 312.527,Z 311.676,A -85,B 0,C 180,E1 -15710.4,E2 -15710.4} C_VEL
LIN {X 0,Y 313.902,Z 317,A -85,B 0,C 180,E1 -15712.248,E2 -15712.248} C_VEL
LIN {X 0,Y 322.134,Z 334.025,A -85,B 0,C 180,E1 -15713.583,E2 -15713.583} C_VEL
LIN {X 0,Y 328.105,Z 348.173,A -85,B 0,C 180,E1 -15714.542,E2 -15714.542} C_VEL
LIN {X 0,Y 328.266,Z 351.78,A -85,B 0,C 180,E1 -15714.647,E2 -15714.647} C_VEL
LIN {X 0,Y 326.079,Z 423.97,A -85,B 0,C 180,E1 -15716.243,E2 -15716.243} C_VEL
LIN {X 0,Y 325.195,Z 437.563,A -85,B 0,C 180,E1 -15716.789,E2 -15716.789} C_VEL
LIN {X 0,Y 324.267,Z 449.709,A -85,B 0,C 180,E1 -15717.536,E2 -15717.536} C_VEL
LIN {X 0,Y 322.898,Z 461.575,A -85,B 0,C 180,E1 -15718.508,E2 -15718.508} C_VEL
LIN {X 0,Y 321.249,Z 473.438,A -85,B 0,C 180,E1 -15719.79,E2 -15719.79} C_VEL
LIN {X 0,Y 319.714,Z 482.954,A -85,B 0,C 180,E1 -15721.078,E2 -15721.078} C_VEL
LIN {X 0,Y 317.953,Z 492.652,A -85,B 0,C 180,E1 -15722.699,E2 -15722.699} C_VEL
LIN {X 0,Y 316.058,Z 501.901,A -85,B 0,C 180,E1 -15724.656,E2 -15724.656} C_VEL
LIN {X 0,Y 314.608,Z 509.31,A -85,B 0,C 180,E1 -15726.639,E2 -15726.639} C_VEL
LIN {X 0,Y 313.547,Z 514.273,A -85,B 0,C 180,E1 -15728.294,E2 -15728.294} C_VEL
LIN {X 0,Y 312.542,Z 519.056,A -85,B 0,C 180,E1 -15730.287,E2 -15730.287} C_VEL
LIN {X 0,Y 311.774,Z 522.675,A -85,B 0,C 180,E1 -15732.282,E2 -15732.282} C_VEL
LIN {X 0,Y 311.229,Z 525.239,A -85,B 0,C 180,E1 -15734.277,E2 -15734.277} C_VEL
LIN {X 0,Y 310.946,Z 526.888,A -85,B 0,C 180,E1 -15736.381,E2 -15736.381} C_VEL
LIN {X 0,Y 310.724,Z 527.477,A -85,B 0,C 180,E1 -15738.254,E2 -15738.254} C_VEL
LIN {X 0,Y 310.592,Z 527.42,A -85,B 0,C 180,E1 -15739.57,E2 -15739.57} C_VEL
LIN {X 0,Y 310.631,Z 526.957,A -85,B 0,C 180,E1 -15740.887,E2 -15740.887} C_VEL
LIN {X 0,Y 310.715,Z 526.056,A -85,B 0,C 180,E1 -15742.2,E2 -15742.2} C_VEL
LIN {X 0,Y 310.935,Z 524.188,A -85,B 0,C 180,E1 -15744.001,E2 -15744.001} C_VEL
LIN {X 0,Y 311.087,Z 520.926,A -85,B 0,C 180,E1 -15746.113,E2 -15746.113} C_VEL
LIN {X 0,Y 311.49,Z 516.83,A -85,B 0,C 180,E1 -15748.06,E2 -15748.06} C_VEL
LIN {X 0,Y 312.068,Z 510.578,A -85,B 0,C 180,E1 -15750.322,E2 -15750.322} C_VEL
LIN {X 0,Y 312.988,Z 503.759,A -85,B 0,C 180,E1 -15752.251,E2 -15752.251} C_VEL
LIN {X 0,Y 313.811,Z 496.817,A -85,B 0,C 180,E1 -15753.852,E2 -15753.852} C_VEL
LIN {X 0,Y 314.772,Z 488.471,A -85,B 0,C 180,E1 -15755.444,E2 -15755.444} C_VEL
LIN {X 0,Y 315.955,Z 478.164,A -85,B 0,C 180,E1 -15757.026,E2 -15757.026} C_VEL
LIN {X 0,Y 317.187,Z 467.934,A -85,B 0,C 180,E1 -15758.28,E2 -15758.28} C_VEL
LIN {X 0,Y 318.203,Z 458.506,A -85,B 0,C 180,E1 -15759.213,E2 -15759.213} C_VEL
LIN {X 0,Y 319.01,Z 446.623,A -85,B 0,C 180,E1 -15760.15,E2 -15760.15} C_VEL
LIN {X 0,Y 319.557,Z 433.716,A -85,B 0,C 180,E1 -15760.894,E2 -15760.894} C_VEL
LIN {X 0,Y 320.293,Z 420.604,A -85,B 0,C 180,E1 -15761.349,E2 -15761.349} C_VEL
LIN {X 0,Y 321.868,Z 345.521,A -85,B 0,C 180,E1 -15763.013,E2 -15763.013} C_VEL
